RoboDK station: 15_holes_program_with_paths.rdk

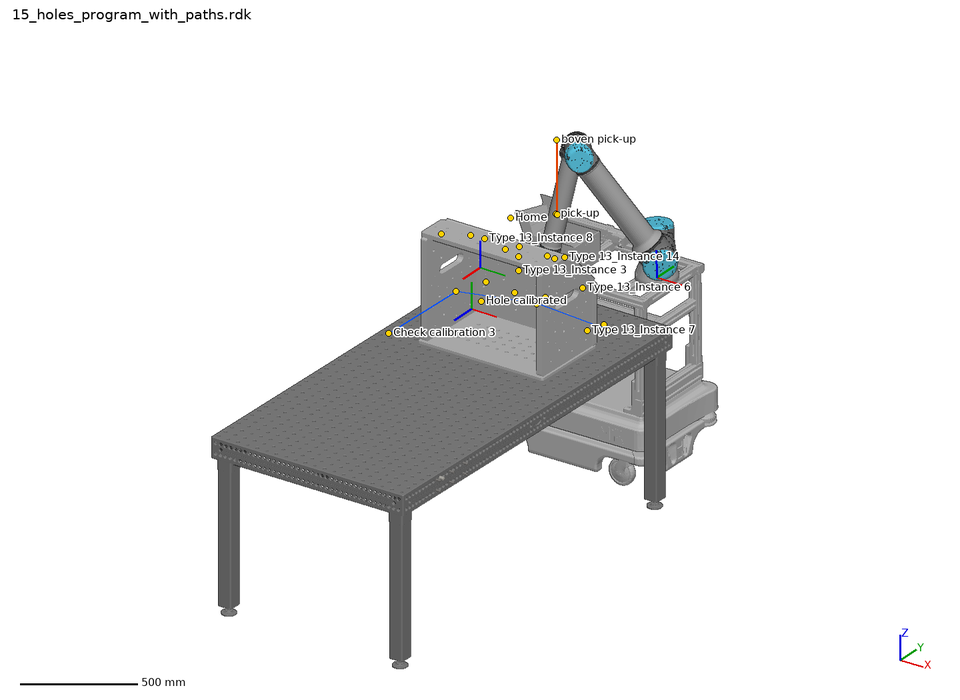
[picture v0: the station drawn from its stored meshes, robots at their saved joint values, targets as dots, program paths as lines]
Station 15_holes_program_with_paths (saved by RoboDK 5.7.0). Poses are relative to the parent item; angles as X-Y-Z fixed-axis rotations.
Station parameters (name, value as stored): 0.4, 1, 1, CollisionFreePlanner, UR10e, CollisionFreePlanner-Rob UR10e, Simplify-Mesh-Settings
  - object Lastafel at (0, 0, 0) mm, size 1021.8 x 2000 x 842 mm
  - object Lastafel_simplified at (0, 0, 0) mm, size 1000 x 2000 x 802.1 mm
  - frame UR10e Base at (-300.71, 2160.25, 91.6) mm, rotated rx 0.6 ry -0.16 rz 0.46 deg
    - robot UR10e: 6 axes, payload 10 kg, reach 1300 mm, repeatability 0.05 mm, weight 28.9 kg
        modified DH rows (alpha deg, a mm, theta deg, d mm): 0, 0, 0, 180.7; 90, 0, 180, 0; 0, 612.6, 0, 0; 0, 571.335, 0, 174.15; -90, 0, 0, 119.85; 90, 0, 180, 116.55
        joint limits [-70, -140, 0, -220, -180, -280] to [85, 0, 170, 200, 180, 115]; home [30.872, -95.296, 116.362, -22.187, 121.11, 179.827]; saved at [38.401, -56.267, 133.515, -77.437, 128.806, 0.409]
      - tool Screwdriver indraaitool, TCP at (215, -0.23, 99.66) mm, rotated rx 0 ry 90 rz 0 deg, size 345 x 117.4 x 144.9 mm, geometry from 0 Screwdriver assembly.STEP
      - tool Camera, TCP at (304, 50.7, 13.6) mm, rotated rx 0 ry 90 rz 0 deg
      - tool pointer, TCP at (196, -0.23, 99.66) mm, rotated rx 0 ry 90 rz 0 deg
      - tool Screwdriver simplified, TCP at (0, 0, 220) mm, size 159.8 x 129.1 x 379.7 mm, geometry from Screwdriver simplified.stl
      - tool indraaien, TCP at (205, 0.2, 100) mm, rotated rx 0 ry 90 rz 0 deg
    - object Assembly mir + frame aangepast naar ur10e versie 2 at (-733.08, 277.19, -552.66) mm, rotated rx 90 ry 0 rz 0.45 deg, size 901.1 x 1139.6 x 580.4 mm, geometry from Assembly mir + frame aangepast naar ur10e versie 2.STEP
    - object Mir + frame simplified at (-733.08, 277.19, -552.66) mm, rotated rx 90 ry 0 rz 0.45 deg, size 925.7 x 1139.7 x 582 mm
    - target boven pick-up (joint target) at (-657.55, 210.4, 385.42) mm, rotated rx 180 ry -0.01 rz 58.34 deg; joints [-50.868, -81.351, 94.607, -13.692, -19.23, -89.565] of UR10e
    - target pick-up (joint target) at (-663.21, 209.22, 32.36) mm, rotated rx 179.99 ry 0 rz 58.33 deg; joints [-50.468, -67.472, 110.452, -43.416, -18.832, -89.554] of UR10e
    - target unclamped (joint target) at (-658.69, 209.89, 32.4) mm, rotated rx -180 ry 0 rz 58.34 deg; joints [-50.794, -47.979, 113.128, 114.877, 19.182, -270.008] of UR10e
  - frame Hoek lastafel at (-1020, 1876.5, 50) mm, rotated rx 0 ry 0 rz -90 deg
    - frame CSV Frame at (350, 200, 0) mm, rotated rx 90 ry 0 rz 90 deg
      - object Test object at (0, 0.01, 0) mm, size 650 x 517 x 400 mm, geometry from Test object.STEP
      - object Test object simplified at (0, 0.01, 0) mm, size 650.1 x 517 x 436.5 mm
      - frame Type 13 at (0, 0, 0) mm
        - target Hole calibrated (Cartesian target) at (50, 50, 0) mm; joints [38.401, -56.267, 133.515, -77.437, 128.806, 0.409] of UR10e
        - target Type 13_Instance 2 (Cartesian target) at (224.21, 141.91, 0) mm, rotated rx 0 ry 0 rz 120 deg; joints [21.978, -61.024, 129.364, 49.468, 78.603, 19.537] of UR10e
        - target Type 13_Instance 3 (Cartesian target) at (246.01, 251.55, 0) mm, rotated rx 0 ry 0 rz 80 deg; joints [29.991, -83.076, 133.126, 30.949, 94.737, 30.232] of UR10e
        - target Type 13_Instance 5 (Cartesian target) at (382.2, 163.02, 0) mm, rotated rx 0 ry 0 rz 100 deg; joints [40.216, -73.928, 140.296, 30.8, 83.246, 40.29] of UR10e
        - target Type 13_Instance 6 (Cartesian target) at (577.65, 261.77, 0) mm, rotated rx 0 ry 0 rz 80 deg; joints [83.526, -84.373, 135.629, 37.157, 100.147, 84.01] of UR10e
        - target Type 13_Instance 7 (Cartesian target) at (602.84, 67, 0) mm, rotated rx 0 ry 0 rz 140 deg; joints [61.233, -52.023, 142.726, 28.243, 47.512, 50] of UR10e
        - target Type 13_Instance 8 (Cartesian target) at (128.87, 405.62, 85.34) mm, rotated rx 0 ry 45 rz -90 deg; joints [24.723, -96.328, 122.329, -93.279, 50.619, -33.648] of UR10e
        - target Type 13_Instance 10 (Cartesian target) at (325.68, 432.59, 112.3) mm, rotated rx 0 ry 45 rz -90 deg; joints [39.423, -108.608, 126.743, -75.897, 57.444, -49.793] of UR10e
        - target Type 13_Instance 12 (Cartesian target) at (502.06, 421.99, 101.71) mm, rotated rx 0 ry 45 rz -90 deg; joints [56.925, -115.887, 130.806, -65.302, 67.776, -65.755] of UR10e
        - target Type 13_Instance 13 (Cartesian target) at (570.16, 369.5, 49.22) mm, rotated rx 0 ry 45 rz -90 deg; joints [62.403, -121.656, 138.779, -65.954, 71.328, -70.219] of UR10e
        - target Type 13_Instance 14 (Cartesian target) at (588.54, 468.7, 148.42) mm, rotated rx 0 ry 45 rz -90 deg; joints [71.01, -111.335, 122.877, -58.584, 77.085, -76.834] of UR10e
        - target Type 13_Instance 15 (Cartesian target) at (192.89, 517, 279.7) mm, rotated rx 0 ry 90 rz -90 deg; joints [52.145, -62.069, 43.009, 18.396, 52.67, -89.759] of UR10e
        - target Type 13_Instance 16 (Cartesian target) at (83.93, 517, 343.03) mm, rotated rx 90 ry 80 rz 0 deg; joints [50.032, -46.238, 16.171, 29.419, 60.538, -89.707] of UR10e
        - target Type 13_Instance 17 (Cartesian target) at (391.06, 517, 308.3) mm, rotated rx 0 ry 90 rz -90 deg; joints [65.267, -66.64, 49.834, 16.228, 65.797, -89.935] of UR10e
        - target Type 13_Instance 18 (Cartesian target) at (577.65, 517, 262.67) mm, rotated rx 0 ry 90 rz -90 deg; joints [77.626, -73.739, 59.711, 13.488, 78.165, -90.075] of UR10e
        - target Type 13_Instance 19 (Cartesian target) at (479.58, 517, 336.9) mm, rotated rx 0 ry 90 rz -90 deg; joints [71.94, -64.785, 47.115, 17.114, 72.467, -90.001] of UR10e
    - target Camera -90 (Cartesian target) at (100, 100, 0) mm, rotated rx 180 ry 0 rz 90 deg; joints [15.382, -77.593, 120.955, -43.48, 105.947, -89.524] of UR10e
    - target Camera +90 (Cartesian target) at (100, 100, 0) mm, rotated rx -180 ry 0 rz -90 deg; joints [17.251, -55.937, 87.569, -31.877, -72.203, -90.48] of UR10e
    - target Camera Calibration (Cartesian target) at (100, 100, 0) mm, rotated rx -180 ry 0 rz 180 deg; joints [5.018, -68.171, 107.665, -44.191, 5.596, -85.486] of UR10e
    - target Camera 2 (Cartesian target) at (150, 750, 0) mm, rotated rx 180 ry 0 rz 180 deg; joints [50.749, -60.173, 157.418, 81.984, -51.264, -269.754] of UR10e
    - target Check calibration 0 (Cartesian target) at (200, 800, 10) mm, rotated rx 180 ry 0 rz 180 deg; joints [69.087, -96.044, 157.848, -62.324, 69.685, -90.102] of UR10e
    - target Check calibration 1 (Cartesian target) at (150, 400, 2) mm, rotated rx 180 ry 0 rz 180 deg; joints [4.739, -84.216, 147.782, -67.962, 5.34, -85.787] of UR10e
    - target Check calibration 2 (Cartesian target) at (250, 50, 2) mm, rotated rx 180 ry 0 rz 180 deg; joints [9.934, -58.947, 106.867, -51.902, 9.691, -86.238] of UR10e
    - target Check calibration 3 (Cartesian target) at (750, 50, 2) mm, rotated rx 180 ry 0 rz 180 deg; joints [40.424, -35.05, 60.293, -26.389, 40.152, -89.277] of UR10e
    - target Home (Cartesian target) at (200, 300, 400) mm, rotated rx 180 ry 0 rz 180 deg; joints [9.713, -85.986, 130.341, 132.467, -10.3, 92.957] of UR10e
  - program Check XY-calibration (7 instructions, listed below)
  - program bovenpickupToType13Instance2 (10 instructions, listed below)
  - program bovenpickupToType13Instance3 (10 instructions, listed below)
  - program bovenpickupToType13Instance5 (11 instructions, listed below)
  - program bovenpickupToType13Instance6 (10 instructions, listed below)
  - program bovenpickupToType13Instance7 (10 instructions, listed below)
  - program bovenpickupToType13Instance8 (12 instructions, listed below)
  - program bovenpickupToType13Instance10 (12 instructions, listed below)
  - program bovenpickupToType13Instance12 (13 instructions, listed below)
  - program bovenpickupToType13Instance13 (13 instructions, listed below)
  - program bovenpickupToType13Instance14 (16 instructions, listed below)
  - program bovenpickupToType13Instance15 (9 instructions, listed below)
  - program bovenpickupToType13Instance16 (13 instructions, listed below)
  - program bovenpickupToType13Instance17 (10 instructions, listed below)
  - program bovenpickupToType13Instance18 (11 instructions, listed below)
  - program bovenpickupToType13Instance19 (11 instructions, listed below)
  - program Type13Instance2Tobovenpickup (11 instructions, listed below)
  - program Type13Instance3Tobovenpickup (10 instructions, listed below)
  - program Type13Instance5Tobovenpickup (12 instructions, listed below)
  - program Type13Instance6Tobovenpickup (10 instructions, listed below)
  - program Type13Instance7Tobovenpickup (12 instructions, listed below)
  - program Type13Instance8Tobovenpickup (14 instructions, listed below)
  - program Type13Instance10Tobovenpickup (11 instructions, listed below)
  - program Type13Instance12Tobovenpickup (12 instructions, listed below)
  - program Type13Instance13Tobovenpickup (11 instructions, listed below)
  - program Type13Instance14Tobovenpickup (11 instructions, listed below)
  - program Type13Instance15Tobovenpickup (9 instructions, listed below)
  - program Type13Instance16Tobovenpickup (10 instructions, listed below)
  - program Type13Instance17Tobovenpickup (10 instructions, listed below)
  - program Type13Instance18Tobovenpickup (10 instructions, listed below)
  - program Type13Instance19Tobovenpickup (10 instructions, listed below)
  - program helicoil pickup (9 instructions, listed below)
  - Python program retract shank (listed below)
  - Python program get_helicoil (listed below)
  - Python program Insert helicoil (listed below)
  - Python program pickup helicoil (listed below)
  - Python program Test get screwdriver data (listed below)
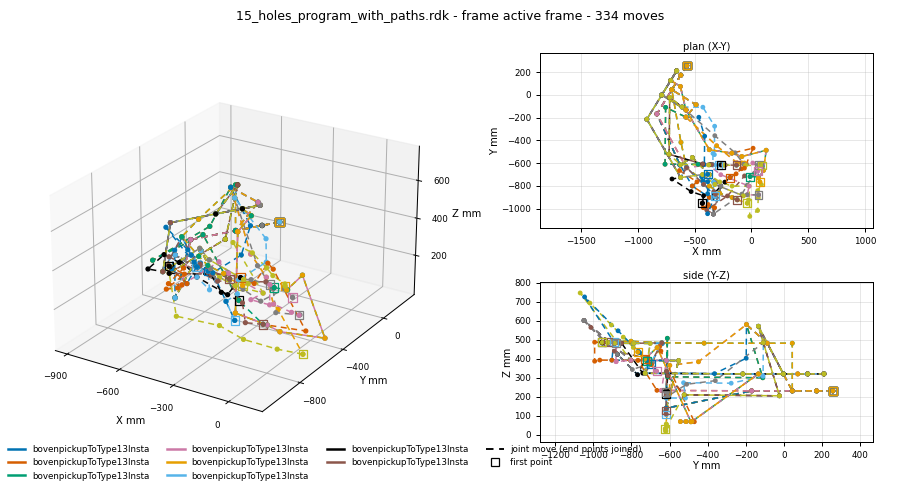
[picture p0: tool path of 15_holes_program_with_paths.rdk in frame active frame, 334 of 342 moves have a stored position in this frame; points joined in program order, loops and branches not executed]
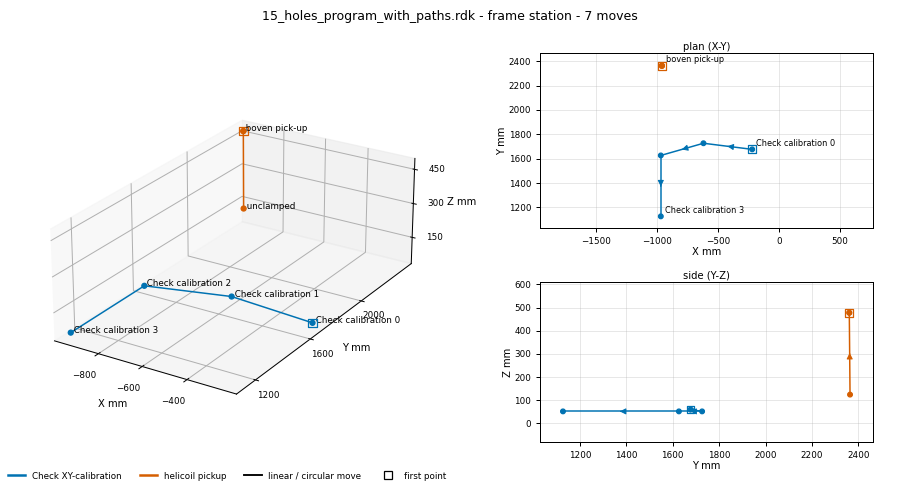
[picture p1: tool path of 15_holes_program_with_paths.rdk in frame station, 7 of 342 moves have a stored position in this frame; points joined in program order, loops and branches not executed]

--- program Check XY-calibration (robot UR10e) ---
  Set Ref.: Hoek lastafel
  Set Tool: pointer
  Set speed (200.0 mm/s)
  MoveL (Check calibration 0)
  MoveL (Check calibration 1)
  MoveL (Check calibration 2)
  MoveL (Check calibration 3)

--- program bovenpickupToType13Instance2 (robot UR10e) ---
  MoveJ (Pt 1 (S642)) to (-569.02, 256.95, 231.44) mm, rotated rx 180 ry -0.01 rz 58.34 deg; joints [-50.868, -81.351, 94.607, -13.692, -19.23, -89.565]
  MoveJ (Pt 2 (S577)) to (-621.5, 171.83, 231.42) mm, rotated rx 180 ry -0.01 rz 58.34 deg; joints [-42.328, -81.409, 94.677, -14.057, -10.69, -89.211]
  MoveJ (Pt 3 (S442)) to (-700.22, 44.15, 231.39) mm, rotated rx 180 ry -0.01 rz 58.34 deg; joints [-29.369, -77.97, 90.586, -9.022, 2.264, -93.593]
  MoveJ (Pt 4 (S421)) to (-487.45, -87.1, 481.39) mm, rotated rx 180 ry -0.01 rz 58.34 deg; joints [-28.022, -101.389, 88.85, 14.844, 3.631, -92.304]
  MoveJ (Pt 5 (S124)) to (-576.74, -196.35, 579.46) mm, rotated rx 89.55 ry -40 rz 0.16 deg; joints [-35.971, -95.179, 103.829, 37.546, 63.204, -24.789]
  MoveJ (Pt 6 (S114)) to (-462.71, -197.66, 402.38) mm, rotated rx 88.03 ry -79.99 rz 1.82 deg; joints [-40.872, -92.425, 119.324, 55.78, 83.328, -40.3]
  MoveJ (Pt 7 (S42)) to (-411.56, -364.05, 321.78) mm, rotated rx -88.79 ry -60.15 rz 178.37 deg; joints [-15.974, -82.156, 125.219, 76.084, 97.176, -13.671]
  MoveJ (Pt 8 (S10)) to (-414.11, -614.03, 324.41) mm, rotated rx -88.79 ry -60.15 rz 178.37 deg; joints [16.405, -73.929, 114.079, 78.537, 81.219, 14.568]
  MoveJ (Pt 9 (S23)) to (-339.48, -616.15, 194.31) mm, rotated rx -88.79 ry -60.15 rz 178.37 deg; joints [19.42, -67.896, 124.439, 61.697, 79.797, 17.249]
  MoveJ (Pt 10 (S33)) to (-289.72, -617.57, 107.58) mm, rotated rx -88.79 ry -60.15 rz 178.37 deg; joints [21.978, -61.024, 129.364, 49.468, 78.603, 19.537]

--- program bovenpickupToType13Instance3 (robot UR10e) ---
  MoveJ (Pt 1 (S258)) to (-569.02, 256.95, 231.44) mm, rotated rx 180 ry -0.01 rz 58.34 deg; joints [-50.868, -81.351, 94.607, -13.692, -19.23, -89.565]
  MoveJ (Pt 2 (S259)) to (-621.5, 171.83, 231.42) mm, rotated rx 180 ry -0.01 rz 58.34 deg; joints [-42.328, -81.409, 94.677, -14.057, -10.69, -89.211]
  MoveJ (Pt 3 (S230)) to (-700.22, 44.15, 231.39) mm, rotated rx 180 ry -0.01 rz 58.34 deg; joints [-29.369, -77.97, 90.586, -9.022, 2.264, -93.593]
  MoveJ (Pt 4 (S386)) to (-487.45, -87.1, 481.39) mm, rotated rx 180 ry -0.01 rz 58.34 deg; joints [-28.022, -101.389, 88.85, 14.844, 3.631, -92.304]
  MoveJ (Pt 5 (S758)) to (-576.74, -196.35, 579.46) mm, rotated rx 89.55 ry -40 rz 0.16 deg; joints [-35.971, -95.179, 103.829, 37.546, 63.204, -24.789]
  MoveJ (Pt 6 (S704)) to (-754.66, -110.75, 300.04) mm, rotated rx 86.59 ry -79.83 rz 2.77 deg; joints [-30.172, -60.169, 89.434, 52.244, 84.533, -29.177]
  MoveJ (Pt 7 (S702)) to (-759.76, -610.7, 305.28) mm, rotated rx 86.59 ry -79.83 rz 2.77 deg; joints [10.723, -56.863, 83.085, 53.769, 91.432, 11.188]
  MoveJ (Pt 8 (S856)) to (-469.6, -611.54, 507.29) mm, rotated rx 86.59 ry -79.83 rz 2.77 deg; joints [17.574, -86.724, 101.894, 65.055, 92.657, 17.965]
  MoveJ (Pt 9 (S864)) to (-348.42, -614.6, 333.21) mm, rotated rx 86.59 ry -79.83 rz 2.77 deg; joints [23.724, -87.864, 122.531, 45.887, 93.715, 24.039]
  MoveJ (Pt 10 (S846)) to (-267.62, -616.65, 217.16) mm, rotated rx 86.59 ry -79.83 rz 2.77 deg; joints [29.991, -83.076, 133.126, 30.949, 94.737, 30.232]

--- program bovenpickupToType13Instance5 (robot UR10e) ---
  MoveJ (Pt 1 (S221)) to (-569.02, 256.95, 231.44) mm, rotated rx 180 ry -0.01 rz 58.34 deg; joints [-50.868, -81.351, 94.607, -13.692, -19.23, -89.565]
  MoveJ (Pt 2 (S222)) to (-621.5, 171.83, 231.42) mm, rotated rx 180 ry -0.01 rz 58.34 deg; joints [-42.328, -81.409, 94.677, -14.057, -10.69, -89.211]
  MoveJ (Pt 3 (S200)) to (-700.22, 44.15, 231.39) mm, rotated rx 180 ry -0.01 rz 58.34 deg; joints [-29.369, -77.97, 90.586, -9.022, 2.264, -93.593]
  MoveJ (Pt 4 (S356)) to (-487.45, -87.1, 481.39) mm, rotated rx 180 ry -0.01 rz 58.34 deg; joints [-28.022, -101.389, 88.85, 14.844, 3.631, -92.304]
  MoveJ (Pt 5 (S742)) to (-576.74, -196.35, 579.46) mm, rotated rx 89.55 ry -40 rz 0.16 deg; joints [-35.971, -95.179, 103.829, 37.546, 63.204, -24.789]
  MoveJ (Pt 6 (S692)) to (-754.66, -110.75, 300.04) mm, rotated rx 86.59 ry -79.83 rz 2.77 deg; joints [-30.172, -60.169, 89.434, 52.244, 84.533, -29.177]
  MoveJ (Pt 7 (S687)) to (-759.76, -610.7, 305.28) mm, rotated rx 86.59 ry -79.83 rz 2.77 deg; joints [10.723, -56.863, 83.085, 53.769, 91.432, 11.188]
  MoveJ (Pt 8 (S846)) to (-469.6, -611.54, 507.29) mm, rotated rx 86.59 ry -79.83 rz 2.77 deg; joints [17.574, -86.724, 101.894, 65.055, 92.657, 17.965]
  MoveJ (Pt 9 (S855)) to (-348.42, -614.6, 333.21) mm, rotated rx 86.59 ry -79.83 rz 2.77 deg; joints [23.724, -87.864, 122.531, 45.887, 93.715, 24.039]
  MoveJ (Pt 10 (S832)) to (-267.62, -616.65, 217.16) mm, rotated rx 86.59 ry -79.83 rz 2.77 deg; joints [29.991, -83.076, 133.126, 30.949, 94.737, 30.232]
  MoveJ (Pt 11 (S795)) to (-131.68, -618.97, 128.27) mm, rotated rx -86.49 ry -80.13 rz 175.95 deg; joints [40.216, -73.928, 140.296, 30.8, 83.246, 40.29]

--- program bovenpickupToType13Instance6 (robot UR10e) ---
  MoveJ (Pt 1 (S198)) to (-569.02, 256.95, 231.44) mm, rotated rx 180 ry -0.01 rz 58.34 deg; joints [-50.868, -81.351, 94.607, -13.692, -19.23, -89.565]
  MoveJ (Pt 2 (S200)) to (-621.5, 171.83, 231.42) mm, rotated rx 180 ry -0.01 rz 58.34 deg; joints [-42.328, -81.409, 94.677, -14.057, -10.69, -89.211]
  MoveJ (Pt 3 (S176)) to (-700.22, 44.15, 231.39) mm, rotated rx 180 ry -0.01 rz 58.34 deg; joints [-29.369, -77.97, 90.586, -9.022, 2.264, -93.593]
  MoveJ (Pt 4 (S337)) to (-487.45, -87.1, 481.39) mm, rotated rx 180 ry -0.01 rz 58.34 deg; joints [-28.022, -101.389, 88.85, 14.844, 3.631, -92.304]
  MoveJ (Pt 5 (S753)) to (-576.74, -196.35, 579.46) mm, rotated rx 89.55 ry -40 rz 0.16 deg; joints [-35.971, -95.179, 103.829, 37.546, 63.204, -24.789]
  MoveJ (Pt 6 (S927)) to (-306.31, -448.13, 384.07) mm, rotated rx 89.47 ry -50 rz 0.28 deg; joints [-10.312, -118.158, 138.236, 30.476, 83.322, -7.663]
  MoveJ (Pt 7 (S951)) to (-127.46, -598.64, 365.16) mm, rotated rx 89.47 ry -50 rz 0.28 deg; joints [52.736, -103.918, 134.566, 32.325, 120.747, 45.438]
  MoveJ (Pt 8 (S904)) to (-87.05, -599.5, 236.84) mm, rotated rx 88.03 ry -79.99 rz 1.82 deg; joints [51.039, -92.195, 140.398, 35.287, 97.676, 50.753]
  MoveJ (Pt 9 (S953)) to (11.43, -599.82, 219.48) mm, rotated rx 88.03 ry -79.99 rz 1.82 deg; joints [71.326, -88.12, 140.046, 34.604, 99.482, 71.185]
  MoveJ (Pt 10 (S985)) to (64.03, -619.93, 226.49) mm, rotated rx 86.59 ry -79.83 rz 2.77 deg; joints [83.526, -84.373, 135.629, 37.157, 100.147, 84.01]

--- program bovenpickupToType13Instance7 (robot UR10e) ---
  MoveJ (Pt 1 (S624)) to (-569.02, 256.95, 231.44) mm, rotated rx 180 ry -0.01 rz 58.34 deg; joints [-50.868, -81.351, 94.607, -13.692, -19.23, -89.565]
  MoveJ (Pt 2 (S566)) to (-621.5, 171.83, 231.42) mm, rotated rx 180 ry -0.01 rz 58.34 deg; joints [-42.328, -81.409, 94.677, -14.057, -10.69, -89.211]
  MoveJ (Pt 3 (S508)) to (-700.22, 44.15, 231.39) mm, rotated rx 180 ry -0.01 rz 58.34 deg; joints [-29.369, -77.97, 90.586, -9.022, 2.264, -93.593]
  MoveJ (Pt 4 (S484)) to (-487.45, -87.1, 481.39) mm, rotated rx 180 ry -0.01 rz 58.34 deg; joints [-28.022, -101.389, 88.85, 14.844, 3.631, -92.304]
  MoveJ (Pt 5 (S95)) to (-576.74, -196.35, 579.46) mm, rotated rx 89.55 ry -40 rz 0.16 deg; joints [-35.971, -95.179, 103.829, 37.546, 63.204, -24.789]
  MoveJ (Pt 6 (S69)) to (-306.31, -448.13, 384.07) mm, rotated rx 89.47 ry -50 rz 0.28 deg; joints [-10.312, -118.158, 138.236, 30.476, 83.322, -7.663]
  MoveJ (Pt 7 (S117)) to (-127.46, -598.64, 365.16) mm, rotated rx 89.47 ry -50 rz 0.28 deg; joints [52.736, -103.918, 134.566, 32.325, 120.747, 45.438]
  MoveJ (Pt 8 (S81)) to (-87.05, -599.5, 236.84) mm, rotated rx 88.03 ry -79.99 rz 1.82 deg; joints [51.039, -92.195, 140.398, 35.287, 97.676, 50.753]
  MoveJ (Pt 9 (S67)) to (-61.73, -599.68, 215.66) mm, rotated rx -0.06 ry -89.66 rz 89.93 deg; joints [51.732, -89.449, 141.404, 37.841, 89.906, 51.849]
  MoveJ (Pt 10 (S129)) to (88.68, -622.23, 31.67) mm, rotated rx -89.21 ry -40.15 rz 178.91 deg; joints [61.233, -52.023, 142.726, 28.243, 47.512, 50]

--- program bovenpickupToType13Instance8 (robot UR10e) ---
  MoveJ (Pt 1 (S440)) to (-569.02, 256.95, 231.44) mm, rotated rx 180 ry -0.01 rz 58.34 deg; joints [-50.868, -81.351, 94.607, -13.692, -19.23, -89.565]
  MoveJ (Pt 2 (S437)) to (-621.5, 171.83, 231.42) mm, rotated rx 180 ry -0.01 rz 58.34 deg; joints [-42.328, -81.409, 94.677, -14.057, -10.69, -89.211]
  MoveJ (Pt 3 (S490)) to (-700.22, 44.15, 231.39) mm, rotated rx 180 ry -0.01 rz 58.34 deg; joints [-29.369, -77.97, 90.586, -9.022, 2.264, -93.593]
  MoveJ (Pt 4 (S533)) to (-831.43, -168.65, 231.34) mm, rotated rx 180 ry -0.01 rz 58.34 deg; joints [-10.139, -68.333, 77.878, -9.215, 21.482, -90.324]
  MoveJ (Pt 5 (S587)) to (-628.82, -616.83, 140.7) mm, rotated rx 180 ry 0.34 rz 89.87 deg; joints [23.562, -63.896, 80.895, -17.582, 23.654, -89.485]
  MoveJ (Pt 6 (S610)) to (-519.72, -552.25, 390.32) mm, rotated rx 180 ry 0.34 rz 89.87 deg; joints [22.274, -79.112, 75.978, 2.531, 22.373, -89.461]
  MoveJ (Pt 7 (S617)) to (-370.06, -702.58, 391.22) mm, rotated rx 180 ry 0.34 rz 89.87 deg; joints [39.494, -78.996, 75.747, 2.876, 39.592, -89.745]
  MoveJ (Pt 8 (S629)) to (-270.28, -802.8, 391.81) mm, rotated rx 180 ry 0.34 rz 89.87 deg; joints [50.999, -75.487, 71.344, 3.823, 51.092, -89.834]
  MoveJ (Pt 9 (S393)) to (-334.84, -1048.74, 600.68) mm, rotated rx 180 ry 45.34 rz 89.87 deg; joints [50.594, -75.677, 73.548, -50.385, 63.524, -59.847]
  MoveJ (Pt 10 (S181)) to (-334.45, -873.03, 422.85) mm, rotated rx 180 ry 45.34 rz 89.87 deg; joints [41.069, -88.108, 106.775, -75.506, 58, -50.992]
  MoveJ (Pt 11 (S109)) to (-334.21, -767.6, 316.15) mm, rotated rx 180 ry 45.34 rz 89.87 deg; joints [33.25, -91.757, 123.172, -92.767, 53.974, -42.917]
  MoveJ (Pt 12 (S94)) to (-385.19, -699.16, 372.43) mm, rotated rx -179.78 ry 45.6 rz 89.57 deg; joints [24.723, -96.328, 122.329, -93.279, 50.619, -33.648]

--- program bovenpickupToType13Instance10 (robot UR10e) ---
  MoveJ (Pt 1 (S435)) to (-569.02, 256.95, 231.44) mm, rotated rx 180 ry -0.01 rz 58.34 deg; joints [-50.868, -81.351, 94.607, -13.692, -19.23, -89.565]
  MoveJ (Pt 2 (S375)) to (-621.5, 171.83, 231.42) mm, rotated rx 180 ry -0.01 rz 58.34 deg; joints [-42.328, -81.409, 94.677, -14.057, -10.69, -89.211]
  MoveJ (Pt 3 (S354)) to (-700.22, 44.15, 231.39) mm, rotated rx 180 ry -0.01 rz 58.34 deg; joints [-29.369, -77.97, 90.586, -9.022, 2.264, -93.593]
  MoveJ (Pt 4 (S390)) to (-831.43, -168.65, 231.34) mm, rotated rx 180 ry -0.01 rz 58.34 deg; joints [-10.139, -68.333, 77.878, -9.215, 21.482, -90.324]
  MoveJ (Pt 5 (S468)) to (-628.82, -616.83, 140.7) mm, rotated rx 180 ry 0.34 rz 89.87 deg; joints [23.562, -63.896, 80.895, -17.582, 23.654, -89.485]
  MoveJ (Pt 6 (S551)) to (-519.72, -552.25, 390.32) mm, rotated rx 180 ry 0.34 rz 89.87 deg; joints [22.274, -79.112, 75.978, 2.531, 22.373, -89.461]
  MoveJ (Pt 7 (S554)) to (-370.06, -702.58, 391.22) mm, rotated rx 180 ry 0.34 rz 89.87 deg; joints [39.494, -78.996, 75.747, 2.876, 39.592, -89.745]
  MoveJ (Pt 8 (S563)) to (-270.28, -802.8, 391.81) mm, rotated rx 180 ry 0.34 rz 89.87 deg; joints [50.999, -75.487, 71.344, 3.823, 51.092, -89.834]
  MoveJ (Pt 9 (S276)) to (-334.84, -1048.74, 600.68) mm, rotated rx 180 ry 45.34 rz 89.87 deg; joints [50.594, -75.677, 73.548, -50.385, 63.524, -59.847]
  MoveJ (Pt 10 (S138)) to (-334.45, -873.03, 422.85) mm, rotated rx 180 ry 45.34 rz 89.87 deg; joints [41.069, -88.108, 106.775, -75.506, 58, -50.992]
  MoveJ (Pt 11 (S166)) to (-234.21, -767.82, 316.15) mm, rotated rx 180 ry 45.34 rz 89.87 deg; joints [39.518, -97.83, 127.836, -87.655, 57.153, -49.479]
  MoveJ (Pt 12 (S207)) to (-188.6, -727.86, 399.15) mm, rotated rx -179.78 ry 45.6 rz 89.57 deg; joints [39.423, -108.608, 126.743, -75.897, 57.444, -49.793]

--- program bovenpickupToType13Instance12 (robot UR10e) ---
  MoveJ (Pt 1 (S490)) to (-569.02, 256.95, 231.44) mm, rotated rx 180 ry -0.01 rz 58.34 deg; joints [-50.868, -81.351, 94.607, -13.692, -19.23, -89.565]
  MoveJ (Pt 2 (S451)) to (-621.5, 171.83, 231.42) mm, rotated rx 180 ry -0.01 rz 58.34 deg; joints [-42.328, -81.409, 94.677, -14.057, -10.69, -89.211]
  MoveJ (Pt 3 (S503)) to (-700.22, 44.15, 231.39) mm, rotated rx 180 ry -0.01 rz 58.34 deg; joints [-29.369, -77.97, 90.586, -9.022, 2.264, -93.593]
  MoveJ (Pt 4 (S564)) to (-831.43, -168.65, 231.34) mm, rotated rx 180 ry -0.01 rz 58.34 deg; joints [-10.139, -68.333, 77.878, -9.215, 21.482, -90.324]
  MoveJ (Pt 5 (S627)) to (-628.82, -616.83, 140.7) mm, rotated rx 180 ry 0.34 rz 89.87 deg; joints [23.562, -63.896, 80.895, -17.582, 23.654, -89.485]
  MoveJ (Pt 6 (S652)) to (-519.72, -552.25, 390.32) mm, rotated rx 180 ry 0.34 rz 89.87 deg; joints [22.274, -79.112, 75.978, 2.531, 22.373, -89.461]
  MoveJ (Pt 7 (S659)) to (-370.06, -702.58, 391.22) mm, rotated rx 180 ry 0.34 rz 89.87 deg; joints [39.494, -78.996, 75.747, 2.876, 39.592, -89.745]
  MoveJ (Pt 8 (S674)) to (-270.28, -802.8, 391.81) mm, rotated rx 180 ry 0.34 rz 89.87 deg; joints [50.999, -75.487, 71.344, 3.823, 51.092, -89.834]
  MoveJ (Pt 9 (S406)) to (-334.84, -1048.74, 600.68) mm, rotated rx 180 ry 45.34 rz 89.87 deg; joints [50.594, -75.677, 73.548, -50.385, 63.524, -59.847]
  MoveJ (Pt 10 (S321)) to (-393.48, -1012.72, 564.35) mm, rotated rx 180 ry 45.34 rz 89.87 deg; joints [45.833, -76.136, 78.115, -56.513, 60.695, -55.521]
  MoveJ (Pt 11 (S226)) to (-211.3, -889.58, 439.32) mm, rotated rx 180 ry 45.34 rz 89.87 deg; joints [50.01, -92.787, 108.942, -68.876, 63.158, -59.384]
  MoveJ (Pt 12 (S275)) to (-60.91, -713.35, 402.9) mm, rotated rx 180 ry 45.34 rz 89.87 deg; joints [50.234, -115.862, 129.495, -66.244, 63.307, -59.629]
  MoveJ (Pt 13 (S348)) to (-12.15, -719.18, 387.98) mm, rotated rx -179.78 ry 45.6 rz 89.57 deg; joints [56.925, -115.887, 130.806, -65.302, 67.776, -65.755]

--- program bovenpickupToType13Instance13 (robot UR10e) ---
  MoveJ (Pt 1 (S502)) to (-569.02, 256.95, 231.44) mm, rotated rx 180 ry -0.01 rz 58.34 deg; joints [-50.868, -81.351, 94.607, -13.692, -19.23, -89.565]
  MoveJ (Pt 2 (S497)) to (-621.5, 171.83, 231.42) mm, rotated rx 180 ry -0.01 rz 58.34 deg; joints [-42.328, -81.409, 94.677, -14.057, -10.69, -89.211]
  MoveJ (Pt 3 (S556)) to (-700.22, 44.15, 231.39) mm, rotated rx 180 ry -0.01 rz 58.34 deg; joints [-29.369, -77.97, 90.586, -9.022, 2.264, -93.593]
  MoveJ (Pt 4 (S613)) to (-831.43, -168.65, 231.34) mm, rotated rx 180 ry -0.01 rz 58.34 deg; joints [-10.139, -68.333, 77.878, -9.215, 21.482, -90.324]
  MoveJ (Pt 5 (S672)) to (-628.82, -616.83, 140.7) mm, rotated rx 180 ry 0.34 rz 89.87 deg; joints [23.562, -63.896, 80.895, -17.582, 23.654, -89.485]
  MoveJ (Pt 6 (S701)) to (-519.72, -552.25, 390.32) mm, rotated rx 180 ry 0.34 rz 89.87 deg; joints [22.274, -79.112, 75.978, 2.531, 22.373, -89.461]
  MoveJ (Pt 7 (S705)) to (-370.06, -702.58, 391.22) mm, rotated rx 180 ry 0.34 rz 89.87 deg; joints [39.494, -78.996, 75.747, 2.876, 39.592, -89.745]
  MoveJ (Pt 8 (S722)) to (-270.28, -802.8, 391.81) mm, rotated rx 180 ry 0.34 rz 89.87 deg; joints [50.999, -75.487, 71.344, 3.823, 51.092, -89.834]
  MoveJ (Pt 9 (S435)) to (-334.84, -1048.74, 600.68) mm, rotated rx 180 ry 45.34 rz 89.87 deg; joints [50.594, -75.677, 73.548, -50.385, 63.524, -59.847]
  MoveJ (Pt 10 (S331)) to (-84.45, -873.59, 422.85) mm, rotated rx 180 ry 45.34 rz 89.87 deg; joints [59.234, -97.73, 114.561, -66.365, 68.949, -67.251]
  MoveJ (Pt 11 (S272)) to (-37.47, -795.07, 343.28) mm, rotated rx 180 ry 45.34 rz 89.87 deg; joints [59.221, -104.089, 128.071, -73.512, 68.939, -67.26]
  MoveJ (Pt 12 (S398)) to (25.63, -689.69, 378.76) mm, rotated rx 180 ry 45.34 rz 89.87 deg; joints [59.247, -119.903, 133.427, -63.039, 68.975, -67.299]
  MoveJ (Pt 13 (S436)) to (56.33, -667.94, 334.76) mm, rotated rx -179.78 ry 45.6 rz 89.57 deg; joints [62.403, -121.656, 138.779, -65.954, 71.328, -70.219]

--- program bovenpickupToType13Instance14 (robot UR10e) ---
  MoveJ (Pt 1 (S636)) to (-569.02, 256.95, 231.44) mm, rotated rx 180 ry -0.01 rz 58.34 deg; joints [-50.868, -81.351, 94.607, -13.692, -19.23, -89.565]
  MoveJ (Pt 2 (S579)) to (-621.5, 171.83, 231.42) mm, rotated rx 180 ry -0.01 rz 58.34 deg; joints [-42.328, -81.409, 94.677, -14.057, -10.69, -89.211]
  MoveJ (Pt 3 (S532)) to (-700.22, 44.15, 231.39) mm, rotated rx 180 ry -0.01 rz 58.34 deg; joints [-29.369, -77.97, 90.586, -9.022, 2.264, -93.593]
  MoveJ (Pt 4 (S413)) to (-831.43, -168.65, 231.34) mm, rotated rx 180 ry -0.01 rz 58.34 deg; joints [-10.139, -68.333, 77.878, -9.215, 21.482, -90.324]
  MoveJ (Pt 5 (S470)) to (-628.82, -616.83, 140.7) mm, rotated rx 180 ry 0.34 rz 89.87 deg; joints [23.562, -63.896, 80.895, -17.582, 23.654, -89.485]
  MoveJ (Pt 6 (S573)) to (-519.72, -552.25, 390.32) mm, rotated rx 180 ry 0.34 rz 89.87 deg; joints [22.274, -79.112, 75.978, 2.531, 22.373, -89.461]
  MoveJ (Pt 7 (S576)) to (-370.06, -702.58, 391.22) mm, rotated rx 180 ry 0.34 rz 89.87 deg; joints [39.494, -78.996, 75.747, 2.876, 39.592, -89.745]
  MoveJ (Pt 8 (S593)) to (-279.16, -766.12, 391.6) mm, rotated rx 180 ry 0.34 rz 89.87 deg; joints [48.532, -78.392, 74.978, 3.089, 48.628, -89.822]
  MoveJ (Pt 9 (S651)) to (-170.28, -803.03, 391.82) mm, rotated rx 180 ry 0.34 rz 89.87 deg; joints [57.613, -79.202, 75.935, 2.972, 57.71, -89.885]
  MoveJ (Pt 10 (S740)) to (-20.28, -803.36, 391.82) mm, rotated rx 180 ry 0.34 rz 89.87 deg; joints [69.118, -82.29, 79.557, 2.458, 69.22, -89.954]
  MoveJ (Pt 11 (S665)) to (-14.78, -1068.99, 745.22) mm, rotated rx -179.78 ry 45.6 rz 89.57 deg; joints [72.225, -79.746, 63.029, -30.149, 77.907, -77.653]
  MoveJ (Pt 12 (S660)) to (53.7, -1017.76, 692.01) mm, rotated rx -179.78 ry 45.6 rz 89.57 deg; joints [76.38, -86.273, 75.842, -35.866, 80.759, -80.743]
  MoveJ (Pt 13 (S562)) to (60.07, -905.32, 577.11) mm, rotated rx -179.78 ry 45.6 rz 89.57 deg; joints [74.313, -98.133, 98.844, -47.262, 79.338, -79.258]
  MoveJ (Pt 14 (S517)) to (55.02, -842.85, 513.38) mm, rotated rx -179.78 ry 45.6 rz 89.57 deg; joints [71.837, -104.176, 110.096, -52.832, 77.645, -77.435]
  MoveJ (Pt 15 (S506)) to (87.31, -790.16, 459.16) mm, rotated rx -179.78 ry 45.6 rz 89.57 deg; joints [73.635, -108.918, 118.831, -56.552, 78.877, -78.786]
  MoveJ (Pt 16 (S476)) to (73.98, -766.28, 434.94) mm, rotated rx -179.78 ry 45.6 rz 89.57 deg; joints [71.01, -111.335, 122.877, -58.584, 77.085, -76.834]

--- program bovenpickupToType13Instance15 (robot UR10e) ---
  MoveJ (Pt 1 (S586)) to (-569.02, 256.95, 231.44) mm, rotated rx 180 ry -0.01 rz 58.34 deg; joints [-50.868, -81.351, 94.607, -13.692, -19.23, -89.565]
  MoveJ (Pt 2 (S526)) to (-621.5, 171.83, 231.42) mm, rotated rx 180 ry -0.01 rz 58.34 deg; joints [-42.328, -81.409, 94.677, -14.057, -10.69, -89.211]
  MoveJ (Pt 3 (S493)) to (-700.22, 44.15, 231.39) mm, rotated rx 180 ry -0.01 rz 58.34 deg; joints [-29.369, -77.97, 90.586, -9.022, 2.264, -93.593]
  MoveJ (Pt 4 (S423)) to (-831.43, -168.65, 231.34) mm, rotated rx 180 ry -0.01 rz 58.34 deg; joints [-10.139, -68.333, 77.878, -9.215, 21.482, -90.324]
  MoveJ (Pt 5 (S303)) to (-628.82, -616.83, 140.7) mm, rotated rx 180 ry 0.34 rz 89.87 deg; joints [23.562, -63.896, 80.895, -17.582, 23.654, -89.485]
  MoveJ (Pt 6 (S431)) to (-628.82, -615.34, 390.69) mm, rotated rx 180 ry 0.34 rz 89.87 deg; joints [23.488, -66.086, 58.723, 6.733, 23.569, -89.434]
  MoveJ (Pt 7 (S390)) to (-520.28, -802.24, 391.81) mm, rotated rx 180 ry 0.34 rz 89.87 deg; joints [38.28, -60.592, 50.44, 9.726, 38.353, -89.675]
  MoveJ (Pt 8 (S324)) to (-370.5, -902.58, 392.41) mm, rotated rx 180 ry 0.34 rz 89.87 deg; joints [50.012, -60.823, 50.732, 9.743, 50.085, -89.789]
  MoveJ (Pt 9 (S347)) to (-322.86, -892.99, 485.67) mm, rotated rx -179.85 ry 0.6 rz 89.42 deg; joints [52.145, -62.069, 43.009, 18.396, 52.67, -89.759]

--- program bovenpickupToType13Instance16 (robot UR10e) ---
  MoveJ (Pt 1 (S521)) to (-569.02, 256.95, 231.44) mm, rotated rx 180 ry -0.01 rz 58.34 deg; joints [-50.868, -81.351, 94.607, -13.692, -19.23, -89.565]
  MoveJ (Pt 2 (S472)) to (-621.5, 171.83, 231.42) mm, rotated rx 180 ry -0.01 rz 58.34 deg; joints [-42.328, -81.409, 94.677, -14.057, -10.69, -89.211]
  MoveJ (Pt 3 (S342)) to (-700.22, 44.15, 231.39) mm, rotated rx 180 ry -0.01 rz 58.34 deg; joints [-29.369, -77.97, 90.586, -9.022, 2.264, -93.593]
  MoveJ (Pt 4 (S284)) to (-831.43, -168.65, 231.34) mm, rotated rx 180 ry -0.01 rz 58.34 deg; joints [-10.139, -68.333, 77.878, -9.215, 21.482, -90.324]
  MoveJ (Pt 5 (S181)) to (-570.99, -643.08, 233.72) mm, rotated rx -179.85 ry 0.6 rz 89.42 deg; joints [26.976, -69.099, 78.835, -10.802, 27.531, -89.229]
  MoveJ (Pt 6 (S175)) to (-632.97, -666.16, 234.14) mm, rotated rx -179.95 ry 0.62 rz 79.41 deg; joints [26.784, -65.118, 73.142, -8.884, 37.333, -89.386]
  MoveJ (Pt 7 (S135)) to (-479.15, -765.67, 391.59) mm, rotated rx 180 ry 0.34 rz 89.87 deg; joints [38.044, -66.874, 59.759, 6.703, 38.126, -89.694]
  MoveJ (Pt 8 (S168)) to (-520.28, -802.24, 391.81) mm, rotated rx 180 ry 0.34 rz 89.87 deg; joints [38.28, -60.592, 50.44, 9.726, 38.353, -89.675]
  MoveJ (Pt 9 (S109)) to (-370.5, -902.58, 392.41) mm, rotated rx 180 ry 0.34 rz 89.87 deg; joints [50.012, -60.823, 50.732, 9.743, 50.085, -89.789]
  MoveJ (Pt 10 (S147)) to (-379.6, -965.89, 392.79) mm, rotated rx 180 ry 0.34 rz 89.87 deg; joints [52.117, -52.777, 37.808, 14.617, 52.182, -89.782]
  MoveJ (Pt 11 (S204)) to (-424.15, -993, 386.99) mm, rotated rx -179.85 ry 0.6 rz 89.42 deg; joints [51.045, -45.985, 26.713, 18.574, 51.562, -89.705]
  MoveJ (Pt 12 (S233)) to (-323.88, -992.98, 486.72) mm, rotated rx -179.85 ry 0.6 rz 89.42 deg; joints [55.939, -45.623, 14.997, 29.967, 56.444, -89.768]
  MoveJ (Pt 13 (S232)) to (-432.46, -955.2, 486.62) mm, rotated rx -179.95 ry 0.62 rz 79.41 deg; joints [50.032, -46.238, 16.171, 29.419, 60.538, -89.707]

--- program bovenpickupToType13Instance17 (robot UR10e) ---
  MoveJ (Pt 1 (S537)) to (-569.02, 256.95, 231.44) mm, rotated rx 180 ry -0.01 rz 58.34 deg; joints [-50.868, -81.351, 94.607, -13.692, -19.23, -89.565]
  MoveJ (Pt 2 (S453)) to (-621.5, 171.83, 231.42) mm, rotated rx 180 ry -0.01 rz 58.34 deg; joints [-42.328, -81.409, 94.677, -14.057, -10.69, -89.211]
  MoveJ (Pt 3 (S393)) to (-700.22, 44.15, 231.39) mm, rotated rx 180 ry -0.01 rz 58.34 deg; joints [-29.369, -77.97, 90.586, -9.022, 2.264, -93.593]
  MoveJ (Pt 4 (S389)) to (-700.25, 44.11, 481.39) mm, rotated rx 180 ry -0.01 rz 58.34 deg; joints [-29.33, -78.074, 65.414, 15.651, 2.287, -92.99]
  MoveJ (Pt 5 (S369)) to (-619.87, -418.56, 481.52) mm, rotated rx -179.85 ry 0.6 rz 89.42 deg; joints [9.338, -76.474, 63.541, 10.042, 9.896, -87.311]
  MoveJ (Pt 6 (S464)) to (-570.29, -640.46, 483.71) mm, rotated rx -179.85 ry 0.6 rz 89.42 deg; joints [26.854, -67.916, 51.844, 14.953, 27.39, -89.171]
  MoveJ (Pt 7 (S675)) to (-370.28, -801.98, 491.81) mm, rotated rx 180 ry 0.34 rz 89.87 deg; joints [45.268, -68.448, 51.699, 16.383, 45.344, -89.76]
  MoveJ (Pt 8 (S801)) to (-279.38, -865.51, 492.19) mm, rotated rx 180 ry 0.34 rz 89.87 deg; joints [53.39, -66.86, 49.394, 17.137, 53.462, -89.821]
  MoveJ (Pt 9 (S881)) to (-170.5, -902.43, 492.41) mm, rotated rx 180 ry 0.34 rz 89.87 deg; joints [61.548, -67.173, 49.822, 17.048, 61.621, -89.875]
  MoveJ (Pt 10 (S919)) to (-124.99, -923.62, 485.44) mm, rotated rx -179.85 ry 0.6 rz 89.42 deg; joints [65.267, -66.64, 49.834, 16.228, 65.797, -89.935]

--- program bovenpickupToType13Instance18 (robot UR10e) ---
  MoveJ (Pt 1 (S552)) to (-569.02, 256.95, 231.44) mm, rotated rx 180 ry -0.01 rz 58.34 deg; joints [-50.868, -81.351, 94.607, -13.692, -19.23, -89.565]
  MoveJ (Pt 2 (S463)) to (-621.5, 171.83, 231.42) mm, rotated rx 180 ry -0.01 rz 58.34 deg; joints [-42.328, -81.409, 94.677, -14.057, -10.69, -89.211]
  MoveJ (Pt 3 (S385)) to (-700.22, 44.15, 231.39) mm, rotated rx 180 ry -0.01 rz 58.34 deg; joints [-29.369, -77.97, 90.586, -9.022, 2.264, -93.593]
  MoveJ (Pt 4 (S301)) to (-831.43, -168.65, 231.34) mm, rotated rx 180 ry -0.01 rz 58.34 deg; joints [-10.139, -68.333, 77.878, -9.215, 21.482, -90.324]
  MoveJ (Pt 5 (S475)) to (-570.99, -643.08, 233.72) mm, rotated rx -179.85 ry 0.6 rz 89.42 deg; joints [26.976, -69.099, 78.835, -10.802, 27.531, -89.229]
  MoveJ (Pt 6 (S530)) to (-378.82, -615.9, 390.7) mm, rotated rx 180 ry 0.34 rz 89.87 deg; joints [32.917, -85.112, 82.825, 1.871, 33.024, -89.684]
  MoveJ (Pt 7 (S681)) to (-270.06, -702.8, 391.22) mm, rotated rx 180 ry 0.34 rz 89.87 deg; joints [45.361, -84.322, 81.904, 2.087, 45.466, -89.81]
  MoveJ (Pt 8 (S992)) to (-20.28, -803.36, 391.82) mm, rotated rx 180 ry 0.34 rz 89.87 deg; joints [69.118, -82.29, 79.557, 2.458, 69.22, -89.954]
  MoveJ (Pt 9 (S1008)) to (-38.22, -879.93, 384.74) mm, rotated rx -179.85 ry 0.6 rz 89.42 deg; joints [70.042, -74.799, 71.224, 3.022, 70.59, -90.011]
  MoveJ (Pt 10 (S1088)) to (61.78, -880.95, 384.48) mm, rotated rx -179.85 ry 0.6 rz 89.42 deg; joints [77.61, -75.19, 71.751, 2.901, 78.159, -90.086]
  MoveJ (Pt 11 (S1090)) to (62.05, -879.9, 484.47) mm, rotated rx -179.85 ry 0.6 rz 89.42 deg; joints [77.626, -73.739, 59.711, 13.488, 78.165, -90.075]

--- program bovenpickupToType13Instance19 (robot UR10e) ---
  MoveJ (Pt 1 (S549)) to (-569.02, 256.95, 231.44) mm, rotated rx 180 ry -0.01 rz 58.34 deg; joints [-50.868, -81.351, 94.607, -13.692, -19.23, -89.565]
  MoveJ (Pt 2 (S464)) to (-621.5, 171.83, 231.42) mm, rotated rx 180 ry -0.01 rz 58.34 deg; joints [-42.328, -81.409, 94.677, -14.057, -10.69, -89.211]
  MoveJ (Pt 3 (S397)) to (-700.22, 44.15, 231.39) mm, rotated rx 180 ry -0.01 rz 58.34 deg; joints [-29.369, -77.97, 90.586, -9.022, 2.264, -93.593]
  MoveJ (Pt 4 (S392)) to (-700.25, 44.11, 481.39) mm, rotated rx 180 ry -0.01 rz 58.34 deg; joints [-29.33, -78.074, 65.414, 15.651, 2.287, -92.99]
  MoveJ (Pt 5 (S371)) to (-619.87, -418.56, 481.52) mm, rotated rx -179.85 ry 0.6 rz 89.42 deg; joints [9.338, -76.474, 63.541, 10.042, 9.896, -87.311]
  MoveJ (Pt 6 (S475)) to (-570.29, -640.46, 483.71) mm, rotated rx -179.85 ry 0.6 rz 89.42 deg; joints [26.854, -67.916, 51.844, 14.953, 27.39, -89.171]
  MoveJ (Pt 7 (S684)) to (-370.28, -801.98, 491.81) mm, rotated rx 180 ry 0.34 rz 89.87 deg; joints [45.268, -68.448, 51.699, 16.383, 45.344, -89.76]
  MoveJ (Pt 8 (S805)) to (-279.38, -865.51, 492.19) mm, rotated rx 180 ry 0.34 rz 89.87 deg; joints [53.39, -66.86, 49.394, 17.137, 53.462, -89.821]
  MoveJ (Pt 9 (S896)) to (-170.5, -902.43, 492.41) mm, rotated rx 180 ry 0.34 rz 89.87 deg; joints [61.548, -67.173, 49.822, 17.048, 61.621, -89.875]
  MoveJ (Pt 10 (S943)) to (-124.99, -923.62, 485.44) mm, rotated rx -179.85 ry 0.6 rz 89.42 deg; joints [65.267, -66.64, 49.834, 16.228, 65.797, -89.935]
  MoveJ (Pt 11 (S999)) to (-36.76, -953.12, 485.51) mm, rotated rx -179.85 ry 0.6 rz 89.42 deg; joints [71.94, -64.785, 47.115, 17.114, 72.467, -90.001]

--- program Type13Instance2Tobovenpickup (robot UR10e) ---
  MoveJ (Pt 1 (S1189)) to (-289.72, -617.57, 107.58) mm, rotated rx -88.79 ry -60.15 rz 178.37 deg; joints [27.28, -59.114, 114.207, 61.653, 76.16, 24.363]
  MoveJ (Pt 2 (S1201)) to (-339.48, -616.15, 194.31) mm, rotated rx -88.79 ry -60.15 rz 178.37 deg; joints [24.893, -63.386, 108.48, 72.156, 77.236, 22.181]
  MoveJ (Pt 3 (S1194)) to (-338.46, -516.17, 193.26) mm, rotated rx -88.79 ry -60.15 rz 178.37 deg; joints [14.894, -67.739, 116.253, 70.372, 81.948, 13.221]
  MoveJ (Pt 4 (S1230)) to (-326.21, -526.44, 274.18) mm, rotated rx -88.79 ry -60.15 rz 178.37 deg; joints [16.405, -73.929, 114.079, 78.537, 81.219, 14.568]
  MoveJ (Pt 5 (S1325)) to (-323.66, -276.47, 271.56) mm, rotated rx -88.79 ry -60.15 rz 178.37 deg; joints [-15.974, -82.156, 125.219, 76.084, 97.176, -13.671]
  MoveJ (Pt 6 (S1213)) to (-427.3, -109.3, 308.25) mm, rotated rx 88.03 ry -79.99 rz 1.82 deg; joints [-40.872, -92.425, 119.324, 55.78, 83.328, -40.3]
  MoveJ (Pt 7 (S1130)) to (-609.73, -107.84, 484.59) mm, rotated rx 89.55 ry -40 rz 0.16 deg; joints [-35.971, -95.179, 103.829, 37.546, 63.204, -24.789]
  MoveJ (Pt 8 (S396)) to (-575.98, -133.64, 570.37) mm, rotated rx 180 ry -0.01 rz 58.34 deg; joints [-28.022, -101.389, 88.85, 14.844, 3.631, -92.304]
  MoveJ (Pt 9 (S200)) to (-788.75, -2.39, 320.37) mm, rotated rx 180 ry -0.01 rz 58.34 deg; joints [-29.369, -77.97, 90.586, -9.022, 2.264, -93.593]
  MoveJ (Pt 10 (S218)) to (-710.03, 125.29, 320.4) mm, rotated rx 180 ry -0.01 rz 58.34 deg; joints [-42.328, -81.409, 94.677, -14.057, -10.69, -89.211]
  MoveJ (Pt 11 (S217)) to (-657.55, 210.41, 320.42) mm, rotated rx 180 ry -0.01 rz 58.34 deg; joints [-50.868, -81.351, 94.607, -13.692, -19.23, -89.565]

--- program Type13Instance3Tobovenpickup (robot UR10e) ---
  MoveJ (Pt 1 (S1294)) to (-267.62, -616.65, 217.16) mm, rotated rx 86.59 ry -79.83 rz 2.77 deg; joints [38.095, -81.767, 118.657, 44.846, 95.948, 38.281]
  MoveJ (Pt 2 (S1236)) to (-366.05, -615.46, 234.78) mm, rotated rx 86.59 ry -79.83 rz 2.77 deg; joints [30.962, -77.951, 111.623, 47.407, 94.864, 31.193]
  MoveJ (Pt 3 (S1190)) to (-428.42, -609.29, 311.25) mm, rotated rx 88.03 ry -79.99 rz 1.82 deg; joints [26.887, -78.117, 102.884, 56.217, 94.291, 26.679]
  MoveJ (Pt 4 (S1144)) to (-723.9, -523.05, 210.67) mm, rotated rx 86.59 ry -79.83 rz 2.77 deg; joints [10.723, -56.863, 83.085, 53.769, 91.432, 11.188]
  MoveJ (Pt 5 (S1130)) to (-718.8, -23.1, 205.42) mm, rotated rx 86.59 ry -79.83 rz 2.77 deg; joints [-30.172, -60.169, 89.434, 52.244, 84.533, -29.177]
  MoveJ (Pt 6 (S1084)) to (-609.73, -107.84, 484.59) mm, rotated rx 89.55 ry -40 rz 0.16 deg; joints [-35.971, -95.179, 103.829, 37.546, 63.204, -24.789]
  MoveJ (Pt 7 (S305)) to (-575.98, -133.64, 570.37) mm, rotated rx 180 ry -0.01 rz 58.34 deg; joints [-28.022, -101.389, 88.85, 14.844, 3.631, -92.304]
  MoveJ (Pt 8 (S158)) to (-788.75, -2.39, 320.37) mm, rotated rx 180 ry -0.01 rz 58.34 deg; joints [-29.369, -77.97, 90.586, -9.022, 2.264, -93.593]
  MoveJ (Pt 9 (S164)) to (-710.03, 125.29, 320.4) mm, rotated rx 180 ry -0.01 rz 58.34 deg; joints [-42.328, -81.409, 94.677, -14.057, -10.69, -89.211]
  MoveJ (Pt 10 (S161)) to (-657.55, 210.41, 320.42) mm, rotated rx 180 ry -0.01 rz 58.34 deg; joints [-50.868, -81.351, 94.607, -13.692, -19.23, -89.565]

--- program Type13Instance5Tobovenpickup (robot UR10e) ---
  MoveJ (Pt 1 (S133)) to (-131.68, -618.97, 128.27) mm, rotated rx -86.49 ry -80.13 rz 175.95 deg; joints [43.816, -74.655, 126.219, 45.161, 82.8, 43.896]
  MoveJ (Pt 2 (S93)) to (-230.2, -618.14, 111.17) mm, rotated rx -86.49 ry -80.13 rz 175.95 deg; joints [35.235, -69.52, 121.457, 45.798, 83.865, 35.319]
  MoveJ (Pt 3 (S77)) to (-247.29, -616.93, 209.69) mm, rotated rx -86.49 ry -80.13 rz 175.95 deg; joints [33.896, -76.471, 117.266, 57.083, 84.043, 33.995]
  MoveJ (Pt 4 (S75)) to (-348.42, -614.6, 333.21) mm, rotated rx 86.59 ry -79.83 rz 2.77 deg; joints [31.991, -83.698, 107.246, 57.617, 95.021, 32.221]
  MoveJ (Pt 5 (S49)) to (-428.42, -609.29, 311.25) mm, rotated rx 88.03 ry -79.99 rz 1.82 deg; joints [26.887, -78.117, 102.884, 56.217, 94.291, 26.679]
  MoveJ (Pt 6 (S13)) to (-723.9, -523.05, 210.67) mm, rotated rx 86.59 ry -79.83 rz 2.77 deg; joints [10.723, -56.863, 83.085, 53.769, 91.432, 11.188]
  MoveJ (Pt 7 (S99)) to (-718.8, -23.1, 205.42) mm, rotated rx 86.59 ry -79.83 rz 2.77 deg; joints [-30.172, -60.169, 89.434, 52.244, 84.533, -29.177]
  MoveJ (Pt 8 (S327)) to (-609.73, -107.84, 484.59) mm, rotated rx 89.55 ry -40 rz 0.16 deg; joints [-35.971, -95.179, 103.829, 37.546, 63.204, -24.789]
  MoveJ (Pt 9 (S848)) to (-575.98, -133.64, 570.37) mm, rotated rx 180 ry -0.01 rz 58.34 deg; joints [-28.022, -101.389, 88.85, 14.844, 3.631, -92.304]
  MoveJ (Pt 10 (S877)) to (-788.75, -2.39, 320.37) mm, rotated rx 180 ry -0.01 rz 58.34 deg; joints [-29.369, -77.97, 90.586, -9.022, 2.264, -93.593]
  MoveJ (Pt 11 (S1076)) to (-710.03, 125.29, 320.4) mm, rotated rx 180 ry -0.01 rz 58.34 deg; joints [-42.328, -81.409, 94.677, -14.057, -10.69, -89.211]
  MoveJ (Pt 12 (S1159)) to (-657.55, 210.41, 320.42) mm, rotated rx 180 ry -0.01 rz 58.34 deg; joints [-50.868, -81.351, 94.607, -13.692, -19.23, -89.565]

--- program Type13Instance6Tobovenpickup (robot UR10e) ---
  MoveJ (Pt 1 (S1552)) to (64.03, -619.93, 226.49) mm, rotated rx 86.59 ry -79.83 rz 2.77 deg; joints [79.719, -85.604, 123.467, 49.881, 100.002, 80.15]
  MoveJ (Pt 2 (S1551)) to (63.98, -610.91, 224.43) mm, rotated rx 88.03 ry -79.99 rz 1.82 deg; joints [79.127, -86.375, 124.464, 49.756, 99.857, 79.091]
  MoveJ (Pt 3 (S1550)) to (-67.18, -610.75, 202.29) mm, rotated rx 89.47 ry -50 rz 0.28 deg; joints [74.524, -83.635, 127.662, 33.189, 128.314, 70.315]
  MoveJ (Pt 4 (S1528)) to (-143.56, -510.2, 265.96) mm, rotated rx 89.47 ry -50 rz 0.28 deg; joints [52.736, -103.918, 134.566, 32.325, 120.747, 45.438]
  MoveJ (Pt 5 (S1495)) to (-322.41, -359.68, 284.88) mm, rotated rx 89.47 ry -50 rz 0.28 deg; joints [-10.312, -118.158, 138.236, 30.476, 83.322, -7.663]
  MoveJ (Pt 6 (S1259)) to (-609.73, -107.84, 484.59) mm, rotated rx 89.55 ry -40 rz 0.16 deg; joints [-35.971, -95.179, 103.829, 37.546, 63.204, -24.789]
  MoveJ (Pt 7 (S659)) to (-575.98, -133.64, 570.37) mm, rotated rx 180 ry -0.01 rz 58.34 deg; joints [-28.022, -101.389, 88.85, 14.844, 3.631, -92.304]
  MoveJ (Pt 8 (S426)) to (-788.75, -2.39, 320.37) mm, rotated rx 180 ry -0.01 rz 58.34 deg; joints [-29.369, -77.97, 90.586, -9.022, 2.264, -93.593]
  MoveJ (Pt 9 (S464)) to (-710.03, 125.29, 320.4) mm, rotated rx 180 ry -0.01 rz 58.34 deg; joints [-42.328, -81.409, 94.677, -14.057, -10.69, -89.211]
  MoveJ (Pt 10 (S461)) to (-657.55, 210.41, 320.42) mm, rotated rx 180 ry -0.01 rz 58.34 deg; joints [-50.868, -81.351, 94.607, -13.692, -19.23, -89.565]

--- program Type13Instance7Tobovenpickup (robot UR10e) ---
  MoveJ (Pt 1 (S149)) to (88.68, -622.23, 31.67) mm, rotated rx -89.21 ry -40.15 rz 178.91 deg; joints [54.508, -52.127, 132.503, 43.528, 51.005, 42.429]
  MoveJ (Pt 2 (S80)) to (-52.22, -620.92, 19.72) mm, rotated rx -89.21 ry -40.15 rz 178.91 deg; joints [39.475, -48.224, 127.844, 52.459, 60.292, 28.076]
  MoveJ (Pt 3 (S40)) to (-239.96, -618.99, 20.85) mm, rotated rx -88.79 ry -60.15 rz 178.37 deg; joints [30.052, -53.136, 118.304, 50.936, 74.933, 26.918]
  MoveJ (Pt 4 (S14)) to (-376.45, -617.21, 57.82) mm, rotated rx -88.79 ry -60.15 rz 178.37 deg; joints [23.502, -51.15, 106.698, 61.979, 77.87, 20.902]
  MoveJ (Pt 5 (S60)) to (-624.3, -614.84, 42.76) mm, rotated rx -86.49 ry -80.13 rz 175.95 deg; joints [18.033, -44.355, 85.466, 58.113, 86.348, 18.222]
  MoveJ (Pt 6 (S76)) to (-723.9, -523.05, 210.67) mm, rotated rx 86.59 ry -79.83 rz 2.77 deg; joints [10.723, -56.863, 83.085, 53.769, 91.432, 11.188]
  MoveJ (Pt 7 (S173)) to (-718.8, -23.1, 205.42) mm, rotated rx 86.59 ry -79.83 rz 2.77 deg; joints [-30.172, -60.169, 89.434, 52.244, 84.533, -29.177]
  MoveJ (Pt 8 (S190)) to (-609.73, -107.84, 484.59) mm, rotated rx 89.55 ry -40 rz 0.16 deg; joints [-35.971, -95.179, 103.829, 37.546, 63.204, -24.789]
  MoveJ (Pt 9 (S938)) to (-575.98, -133.64, 570.37) mm, rotated rx 180 ry -0.01 rz 58.34 deg; joints [-28.022, -101.389, 88.85, 14.844, 3.631, -92.304]
  MoveJ (Pt 10 (S960)) to (-788.75, -2.39, 320.37) mm, rotated rx 180 ry -0.01 rz 58.34 deg; joints [-29.369, -77.97, 90.586, -9.022, 2.264, -93.593]
  MoveJ (Pt 11 (S1072)) to (-710.03, 125.29, 320.4) mm, rotated rx 180 ry -0.01 rz 58.34 deg; joints [-42.328, -81.409, 94.677, -14.057, -10.69, -89.211]
  MoveJ (Pt 12 (S1133)) to (-657.55, 210.41, 320.42) mm, rotated rx 180 ry -0.01 rz 58.34 deg; joints [-50.868, -81.351, 94.607, -13.692, -19.23, -89.565]

--- program Type13Instance8Tobovenpickup (robot UR10e) ---
  MoveJ (Pt 1 (S133)) to (-385.19, -699.16, 372.43) mm, rotated rx -179.78 ry 45.6 rz 89.57 deg; joints [27.437, -91.84, 132.735, -106.178, 51.694, -36.835]
  MoveJ (Pt 2 (S138)) to (-438.23, -721.07, 395.91) mm, rotated rx 180 ry 45.34 rz 89.87 deg; joints [26.844, -88.33, 126.117, -103.53, 51.12, -35.687]
  MoveJ (Pt 3 (S174)) to (-425.45, -756.99, 432.24) mm, rotated rx 180 ry 45.34 rz 89.87 deg; joints [30.527, -89.213, 121.956, -95.887, 52.71, -39.909]
  MoveJ (Pt 4 (S192)) to (-385.14, -764.67, 439.92) mm, rotated rx 180 ry 45.34 rz 89.87 deg; joints [33.25, -91.757, 123.172, -92.767, 53.974, -42.917]
  MoveJ (Pt 5 (S285)) to (-385.37, -870.1, 546.62) mm, rotated rx 180 ry 45.34 rz 89.87 deg; joints [41.069, -88.108, 106.775, -75.506, 58, -50.992]
  MoveJ (Pt 6 (S626)) to (-385.77, -1045.81, 724.45) mm, rotated rx 180 ry 45.34 rz 89.87 deg; joints [50.594, -75.677, 73.548, -50.385, 63.524, -59.847]
  MoveJ (Pt 7 (S967)) to (-321.4, -888.21, 481.33) mm, rotated rx 180 ry 0.34 rz 89.87 deg; joints [50.999, -75.487, 71.344, 3.823, 51.092, -89.834]
  MoveJ (Pt 8 (S943)) to (-421.18, -787.99, 480.73) mm, rotated rx 180 ry 0.34 rz 89.87 deg; joints [39.494, -78.996, 75.747, 2.876, 39.592, -89.745]
  MoveJ (Pt 9 (S939)) to (-570.84, -637.66, 479.83) mm, rotated rx 180 ry 0.34 rz 89.87 deg; joints [22.274, -79.112, 75.978, 2.531, 22.373, -89.461]
  MoveJ (Pt 10 (S920)) to (-622.54, -727.68, 323.76) mm, rotated rx -179.85 ry 0.6 rz 89.42 deg; joints [26.976, -69.099, 78.835, -10.802, 27.531, -89.229]
  MoveJ (Pt 11 (S842)) to (-919.96, -215.19, 320.32) mm, rotated rx 180 ry -0.01 rz 58.34 deg; joints [-10.139, -68.333, 77.878, -9.215, 21.482, -90.324]
  MoveJ (Pt 12 (S781)) to (-788.75, -2.39, 320.37) mm, rotated rx 180 ry -0.01 rz 58.34 deg; joints [-29.369, -77.97, 90.586, -9.022, 2.264, -93.593]
  MoveJ (Pt 13 (S715)) to (-710.03, 125.29, 320.4) mm, rotated rx 180 ry -0.01 rz 58.34 deg; joints [-42.328, -81.409, 94.677, -14.057, -10.69, -89.211]
  MoveJ (Pt 14 (S719)) to (-657.55, 210.41, 320.42) mm, rotated rx 180 ry -0.01 rz 58.34 deg; joints [-50.868, -81.351, 94.607, -13.692, -19.23, -89.565]

--- program Type13Instance10Tobovenpickup (robot UR10e) ---
  MoveJ (Pt 1 (S289)) to (-188.6, -727.86, 399.15) mm, rotated rx -179.78 ry 45.6 rz 89.57 deg; joints [44.179, -104.134, 137.124, -88.349, 60.047, -54.438]
  MoveJ (Pt 2 (S334)) to (-134.98, -694.94, 368.79) mm, rotated rx 180 ry 45.34 rz 89.87 deg; joints [46.017, -108.293, 143.092, -89.199, 60.781, -55.795]
  MoveJ (Pt 3 (S487)) to (-88.08, -650.72, 466.2) mm, rotated rx 180 ry 45.34 rz 89.87 deg; joints [46.59, -123.031, 139.305, -70.413, 61.141, -56.34]
  MoveJ (Pt 4 (S556)) to (-62.19, -645.32, 440.42) mm, rotated rx -179.78 ry 45.6 rz 89.57 deg; joints [49.872, -123.512, 142.123, -71.486, 63.406, -59.701]
  MoveJ (Pt 5 (S900)) to (14.21, -469.79, 69.28) mm, rotated rx -179.85 ry 0.6 rz 89.42 deg; joints [50.086, -118.746, 152.354, -34.198, 50.72, -89.874]
  MoveJ (Pt 6 (S751)) to (-172.83, -513.5, 70.26) mm, rotated rx -179.85 ry 0.6 rz 89.42 deg; joints [29.31, -103.236, 144.185, -41.809, 29.916, -89.469]
  MoveJ (Pt 7 (S617)) to (-370.7, -482.88, 70.48) mm, rotated rx -179.85 ry 0.6 rz 89.42 deg; joints [13.149, -90.207, 133.323, -44.907, 13.74, -88.44]
  MoveJ (Pt 8 (S631)) to (-575.95, -133.6, 320.37) mm, rotated rx 180 ry -0.01 rz 58.34 deg; joints [-28.099, -101.276, 114.057, -10.072, 3.57, -92.709]
  MoveJ (Pt 9 (S658)) to (-624.91, 72.81, 320.4) mm, rotated rx 180 ry -0.01 rz 58.34 deg; joints [-44.286, -90.997, 104.968, -14.694, -12.634, -89.275]
  MoveJ (Pt 10 (S644)) to (-710.03, 125.29, 320.4) mm, rotated rx 180 ry -0.01 rz 58.34 deg; joints [-42.328, -81.409, 94.677, -14.057, -10.69, -89.211]
  MoveJ (Pt 11 (S728)) to (-657.55, 210.41, 320.42) mm, rotated rx 180 ry -0.01 rz 58.34 deg; joints [-50.868, -81.351, 94.607, -13.692, -19.23, -89.565]

--- program Type13Instance12Tobovenpickup (robot UR10e) ---
  MoveJ (Pt 1 (S513)) to (-12.15, -719.18, 387.98) mm, rotated rx -179.78 ry 45.6 rz 89.57 deg; joints [63.878, -109.293, 140.39, -79.57, 72.279, -71.376]
  MoveJ (Pt 2 (S634)) to (61.77, -722.18, 395.92) mm, rotated rx 180 ry 45.34 rz 89.87 deg; joints [74.106, -108.805, 138.636, -76.185, 78.931, -78.761]
  MoveJ (Pt 3 (S633)) to (61.39, -730.41, 398.49) mm, rotated rx -179.78 ry 45.6 rz 89.57 deg; joints [74.725, -107.766, 137.885, -76.607, 79.613, -79.609]
  MoveJ (Pt 4 (S805)) to (105.76, -665.07, 458.39) mm, rotated rx -179.78 ry 45.6 rz 89.57 deg; joints [79.214, -118.718, 137.07, -64.344, 82.733, -82.897]
  MoveJ (Pt 5 (S925)) to (129.27, -487.99, 69.16) mm, rotated rx -179.85 ry 0.6 rz 89.42 deg; joints [80.537, -109.201, 147.969, -39.291, 81.151, -90.195]
  MoveJ (Pt 6 (S723)) to (-84.6, -543.01, 70.32) mm, rotated rx -179.85 ry 0.6 rz 89.42 deg; joints [44.503, -103.995, 144.682, -41.32, 45.11, -89.793]
  MoveJ (Pt 7 (S709)) to (-172.83, -513.5, 70.26) mm, rotated rx -179.85 ry 0.6 rz 89.42 deg; joints [29.31, -103.236, 144.185, -41.809, 29.916, -89.469]
  MoveJ (Pt 8 (S570)) to (-370.7, -482.88, 70.48) mm, rotated rx -179.85 ry 0.6 rz 89.42 deg; joints [13.149, -90.207, 133.323, -44.907, 13.74, -88.44]
  MoveJ (Pt 9 (S757)) to (-575.95, -133.6, 320.37) mm, rotated rx 180 ry -0.01 rz 58.34 deg; joints [-28.099, -101.276, 114.057, -10.072, 3.57, -92.709]
  MoveJ (Pt 10 (S706)) to (-624.91, 72.81, 320.4) mm, rotated rx 180 ry -0.01 rz 58.34 deg; joints [-44.286, -90.997, 104.968, -14.694, -12.634, -89.275]
  MoveJ (Pt 11 (S716)) to (-710.03, 125.29, 320.4) mm, rotated rx 180 ry -0.01 rz 58.34 deg; joints [-42.328, -81.409, 94.677, -14.057, -10.69, -89.211]
  MoveJ (Pt 12 (S755)) to (-657.55, 210.41, 320.42) mm, rotated rx 180 ry -0.01 rz 58.34 deg; joints [-50.868, -81.351, 94.607, -13.692, -19.23, -89.565]

--- program Type13Instance13Tobovenpickup (robot UR10e) ---
  MoveJ (Pt 1 (S612)) to (56.33, -667.94, 334.76) mm, rotated rx -179.78 ry 45.6 rz 89.57 deg; joints [70.982, -111.414, 147.715, -83.342, 77.05, -76.836]
  MoveJ (Pt 2 (S623)) to (61.39, -730.41, 398.49) mm, rotated rx -179.78 ry 45.6 rz 89.57 deg; joints [74.725, -107.766, 137.885, -76.607, 79.613, -79.609]
  MoveJ (Pt 3 (S799)) to (105.76, -665.07, 458.39) mm, rotated rx -179.78 ry 45.6 rz 89.57 deg; joints [79.214, -118.718, 137.07, -64.344, 82.733, -82.897]
  MoveJ (Pt 4 (S942)) to (129.27, -487.99, 69.16) mm, rotated rx -179.85 ry 0.6 rz 89.42 deg; joints [80.537, -109.201, 147.969, -39.291, 81.151, -90.195]
  MoveJ (Pt 5 (S777)) to (-84.6, -543.01, 70.32) mm, rotated rx -179.85 ry 0.6 rz 89.42 deg; joints [44.503, -103.995, 144.682, -41.32, 45.11, -89.793]
  MoveJ (Pt 6 (S768)) to (-172.83, -513.5, 70.26) mm, rotated rx -179.85 ry 0.6 rz 89.42 deg; joints [29.31, -103.236, 144.185, -41.809, 29.916, -89.469]
  MoveJ (Pt 7 (S651)) to (-370.7, -482.88, 70.48) mm, rotated rx -179.85 ry 0.6 rz 89.42 deg; joints [13.149, -90.207, 133.323, -44.907, 13.74, -88.44]
  MoveJ (Pt 8 (S852)) to (-575.95, -133.6, 320.37) mm, rotated rx 180 ry -0.01 rz 58.34 deg; joints [-28.099, -101.276, 114.057, -10.072, 3.57, -92.709]
  MoveJ (Pt 9 (S802)) to (-624.91, 72.81, 320.4) mm, rotated rx 180 ry -0.01 rz 58.34 deg; joints [-44.286, -90.997, 104.968, -14.694, -12.634, -89.275]
  MoveJ (Pt 10 (S807)) to (-710.03, 125.29, 320.4) mm, rotated rx 180 ry -0.01 rz 58.34 deg; joints [-42.328, -81.409, 94.677, -14.057, -10.69, -89.211]
  MoveJ (Pt 11 (S809)) to (-657.55, 210.41, 320.42) mm, rotated rx 180 ry -0.01 rz 58.34 deg; joints [-50.868, -81.351, 94.607, -13.692, -19.23, -89.565]

--- program Type13Instance14Tobovenpickup (robot UR10e) ---
  MoveJ (Pt 1 (S656)) to (73.98, -766.28, 434.94) mm, rotated rx -179.78 ry 45.6 rz 89.57 deg; joints [77.62, -105.311, 132.061, -72.899, 81.611, -81.723]
  MoveJ (Pt 2 (S570)) to (61.39, -730.41, 398.49) mm, rotated rx -179.78 ry 45.6 rz 89.57 deg; joints [74.725, -107.766, 137.885, -76.607, 79.613, -79.609]
  MoveJ (Pt 3 (S750)) to (105.76, -665.07, 458.39) mm, rotated rx -179.78 ry 45.6 rz 89.57 deg; joints [79.214, -118.718, 137.07, -64.344, 82.733, -82.897]
  MoveJ (Pt 4 (S864)) to (129.27, -487.99, 69.16) mm, rotated rx -179.85 ry 0.6 rz 89.42 deg; joints [80.537, -109.201, 147.969, -39.291, 81.151, -90.195]
  MoveJ (Pt 5 (S664)) to (-84.6, -543.01, 70.32) mm, rotated rx -179.85 ry 0.6 rz 89.42 deg; joints [44.503, -103.995, 144.682, -41.32, 45.11, -89.793]
  MoveJ (Pt 6 (S644)) to (-172.83, -513.5, 70.26) mm, rotated rx -179.85 ry 0.6 rz 89.42 deg; joints [29.31, -103.236, 144.185, -41.809, 29.916, -89.469]
  MoveJ (Pt 7 (S579)) to (-370.7, -482.88, 70.48) mm, rotated rx -179.85 ry 0.6 rz 89.42 deg; joints [13.149, -90.207, 133.323, -44.907, 13.74, -88.44]
  MoveJ (Pt 8 (S770)) to (-575.95, -133.6, 320.37) mm, rotated rx 180 ry -0.01 rz 58.34 deg; joints [-28.099, -101.276, 114.057, -10.072, 3.57, -92.709]
  MoveJ (Pt 9 (S728)) to (-624.91, 72.81, 320.4) mm, rotated rx 180 ry -0.01 rz 58.34 deg; joints [-44.286, -90.997, 104.968, -14.694, -12.634, -89.275]
  MoveJ (Pt 10 (S814)) to (-710.03, 125.29, 320.4) mm, rotated rx 180 ry -0.01 rz 58.34 deg; joints [-42.328, -81.409, 94.677, -14.057, -10.69, -89.211]
  MoveJ (Pt 11 (S817)) to (-657.55, 210.41, 320.42) mm, rotated rx 180 ry -0.01 rz 58.34 deg; joints [-50.868, -81.351, 94.607, -13.692, -19.23, -89.565]

--- program Type13Instance15Tobovenpickup (robot UR10e) ---
  MoveJ (Pt 1 (S339)) to (-322.86, -892.99, 485.67) mm, rotated rx -179.85 ry 0.6 rz 89.42 deg; joints [51.242, -75.215, 70.66, 3.908, 51.792, -89.787]
  MoveJ (Pt 2 (S307)) to (-330.28, -851.53, 481.11) mm, rotated rx 180 ry 0.34 rz 89.87 deg; joints [48.532, -78.392, 74.978, 3.089, 48.628, -89.822]
  MoveJ (Pt 3 (S206)) to (-421.18, -787.99, 480.73) mm, rotated rx 180 ry 0.34 rz 89.87 deg; joints [39.494, -78.996, 75.747, 2.876, 39.592, -89.745]
  MoveJ (Pt 4 (S80)) to (-570.29, -640.46, 483.71) mm, rotated rx -179.85 ry 0.6 rz 89.42 deg; joints [22.508, -79.344, 75.967, 2.131, 23.068, -89.026]
  MoveJ (Pt 5 (S110)) to (-622.54, -727.68, 323.76) mm, rotated rx -179.85 ry 0.6 rz 89.42 deg; joints [26.976, -69.099, 78.835, -10.802, 27.531, -89.229]
  MoveJ (Pt 6 (S55)) to (-919.96, -215.19, 320.32) mm, rotated rx 180 ry -0.01 rz 58.34 deg; joints [-10.139, -68.333, 77.878, -9.215, 21.482, -90.324]
  MoveJ (Pt 7 (S70)) to (-788.75, -2.39, 320.37) mm, rotated rx 180 ry -0.01 rz 58.34 deg; joints [-29.369, -77.97, 90.586, -9.022, 2.264, -93.593]
  MoveJ (Pt 8 (S104)) to (-710.03, 125.29, 320.4) mm, rotated rx 180 ry -0.01 rz 58.34 deg; joints [-42.328, -81.409, 94.677, -14.057, -10.69, -89.211]
  MoveJ (Pt 9 (S159)) to (-657.55, 210.41, 320.42) mm, rotated rx 180 ry -0.01 rz 58.34 deg; joints [-50.868, -81.351, 94.607, -13.692, -19.23, -89.565]

--- program Type13Instance16Tobovenpickup (robot UR10e) ---
  MoveJ (Pt 1 (S641)) to (-432.46, -955.2, 486.62) mm, rotated rx -179.95 ry 0.62 rz 79.41 deg; joints [50.203, -65.499, 57.33, 7.549, 60.74, -89.765]
  MoveJ (Pt 2 (S593)) to (-430.5, -951.3, 481.71) mm, rotated rx 180 ry 0.34 rz 89.87 deg; joints [47.928, -64.077, 55.644, 8.081, 48.005, -89.782]
  MoveJ (Pt 3 (S498)) to (-421.4, -887.99, 481.33) mm, rotated rx 180 ry 0.34 rz 89.87 deg; joints [45.289, -70.532, 64.83, 5.348, 45.375, -89.777]
  MoveJ (Pt 4 (S476)) to (-530.28, -851.08, 481.11) mm, rotated rx 180 ry 0.34 rz 89.87 deg; joints [38.044, -66.874, 59.759, 6.703, 38.126, -89.694]
  MoveJ (Pt 5 (S248)) to (-698.6, -740.46, 324.1) mm, rotated rx -179.95 ry 0.62 rz 79.41 deg; joints [26.784, -65.118, 73.142, -8.884, 37.333, -89.386]
  MoveJ (Pt 6 (S24)) to (-622.54, -727.68, 323.76) mm, rotated rx -179.85 ry 0.6 rz 89.42 deg; joints [26.976, -69.099, 78.835, -10.802, 27.531, -89.229]
  MoveJ (Pt 7 (S180)) to (-919.96, -215.19, 320.32) mm, rotated rx 180 ry -0.01 rz 58.34 deg; joints [-10.139, -68.333, 77.878, -9.215, 21.482, -90.324]
  MoveJ (Pt 8 (S363)) to (-788.75, -2.39, 320.37) mm, rotated rx 180 ry -0.01 rz 58.34 deg; joints [-29.369, -77.97, 90.586, -9.022, 2.264, -93.593]
  MoveJ (Pt 9 (S405)) to (-710.03, 125.29, 320.4) mm, rotated rx 180 ry -0.01 rz 58.34 deg; joints [-42.328, -81.409, 94.677, -14.057, -10.69, -89.211]
  MoveJ (Pt 10 (S481)) to (-657.55, 210.41, 320.42) mm, rotated rx 180 ry -0.01 rz 58.34 deg; joints [-50.868, -81.351, 94.607, -13.692, -19.23, -89.565]

--- program Type13Instance17Tobovenpickup (robot UR10e) ---
  MoveJ (Pt 1 (S654)) to (-124.99, -923.62, 485.44) mm, rotated rx -179.85 ry 0.6 rz 89.42 deg; joints [66.188, -78.303, 74.533, 3.209, 66.741, -89.976]
  MoveJ (Pt 2 (S587)) to (-315.79, -875.28, 485.47) mm, rotated rx -179.95 ry 0.62 rz 79.41 deg; joints [53.381, -78.315, 74.551, 3.172, 63.935, -89.83]
  MoveJ (Pt 3 (S501)) to (-330.28, -851.53, 481.11) mm, rotated rx 180 ry 0.34 rz 89.87 deg; joints [48.532, -78.392, 74.978, 3.089, 48.628, -89.822]
  MoveJ (Pt 4 (S442)) to (-421.18, -787.99, 480.73) mm, rotated rx 180 ry 0.34 rz 89.87 deg; joints [39.494, -78.996, 75.747, 2.876, 39.592, -89.745]
  MoveJ (Pt 5 (S269)) to (-570.29, -640.46, 483.71) mm, rotated rx -179.85 ry 0.6 rz 89.42 deg; joints [22.508, -79.344, 75.967, 2.131, 23.068, -89.026]
  MoveJ (Pt 6 (S286)) to (-622.54, -727.68, 323.76) mm, rotated rx -179.85 ry 0.6 rz 89.42 deg; joints [26.976, -69.099, 78.835, -10.802, 27.531, -89.229]
  MoveJ (Pt 7 (S341)) to (-919.96, -215.19, 320.32) mm, rotated rx 180 ry -0.01 rz 58.34 deg; joints [-10.139, -68.333, 77.878, -9.215, 21.482, -90.324]
  MoveJ (Pt 8 (S383)) to (-788.75, -2.39, 320.37) mm, rotated rx 180 ry -0.01 rz 58.34 deg; joints [-29.369, -77.97, 90.586, -9.022, 2.264, -93.593]
  MoveJ (Pt 9 (S422)) to (-710.03, 125.29, 320.4) mm, rotated rx 180 ry -0.01 rz 58.34 deg; joints [-42.328, -81.409, 94.677, -14.057, -10.69, -89.211]
  MoveJ (Pt 10 (S468)) to (-657.55, 210.41, 320.42) mm, rotated rx 180 ry -0.01 rz 58.34 deg; joints [-50.868, -81.351, 94.607, -13.692, -19.23, -89.565]

--- program Type13Instance18Tobovenpickup (robot UR10e) ---
  MoveJ (Pt 1 (S720)) to (62.05, -879.9, 484.47) mm, rotated rx -179.85 ry 0.6 rz 89.42 deg; joints [80.496, -83.347, 80.539, 2.274, 81.055, -90.126]
  MoveJ (Pt 2 (S584)) to (-37.94, -878.88, 484.74) mm, rotated rx -179.85 ry 0.6 rz 89.42 deg; joints [71.784, -83.671, 80.876, 2.251, 72.344, -90.042]
  MoveJ (Pt 3 (S506)) to (-71.4, -888.77, 481.33) mm, rotated rx 180 ry 0.34 rz 89.87 deg; joints [69.118, -82.29, 79.557, 2.458, 69.22, -89.954]
  MoveJ (Pt 4 (S121)) to (-321.18, -788.22, 480.73) mm, rotated rx 180 ry 0.34 rz 89.87 deg; joints [45.361, -84.322, 81.904, 2.087, 45.466, -89.81]
  MoveJ (Pt 5 (S91)) to (-429.94, -701.31, 480.21) mm, rotated rx 180 ry 0.34 rz 89.87 deg; joints [32.917, -85.112, 82.825, 1.871, 33.024, -89.684]
  MoveJ (Pt 6 (S68)) to (-622.54, -727.68, 323.76) mm, rotated rx -179.85 ry 0.6 rz 89.42 deg; joints [26.976, -69.099, 78.835, -10.802, 27.531, -89.229]
  MoveJ (Pt 7 (S39)) to (-919.96, -215.19, 320.32) mm, rotated rx 180 ry -0.01 rz 58.34 deg; joints [-10.139, -68.333, 77.878, -9.215, 21.482, -90.324]
  MoveJ (Pt 8 (S16)) to (-788.75, -2.39, 320.37) mm, rotated rx 180 ry -0.01 rz 58.34 deg; joints [-29.369, -77.97, 90.586, -9.022, 2.264, -93.593]
  MoveJ (Pt 9 (S32)) to (-710.03, 125.29, 320.4) mm, rotated rx 180 ry -0.01 rz 58.34 deg; joints [-42.328, -81.409, 94.677, -14.057, -10.69, -89.211]
  MoveJ (Pt 10 (S52)) to (-657.55, 210.41, 320.42) mm, rotated rx 180 ry -0.01 rz 58.34 deg; joints [-50.868, -81.351, 94.607, -13.692, -19.23, -89.565]

--- program Type13Instance19Tobovenpickup (robot UR10e) ---
  MoveJ (Pt 1 (S655)) to (-36.76, -953.12, 485.51) mm, rotated rx -179.85 ry 0.6 rz 89.42 deg; joints [73.751, -76.309, 72.059, 3.706, 74.301, -90.05]
  MoveJ (Pt 2 (S624)) to (-25, -924.64, 485.18) mm, rotated rx -179.85 ry 0.6 rz 89.42 deg; joints [74.025, -79.207, 75.653, 3.013, 74.578, -90.057]
  MoveJ (Pt 3 (S540)) to (-71.4, -888.77, 481.33) mm, rotated rx 180 ry 0.34 rz 89.87 deg; joints [69.118, -82.29, 79.557, 2.458, 69.22, -89.954]
  MoveJ (Pt 4 (S332)) to (-321.18, -788.22, 480.73) mm, rotated rx 180 ry 0.34 rz 89.87 deg; joints [45.361, -84.322, 81.904, 2.087, 45.466, -89.81]
  MoveJ (Pt 5 (S298)) to (-429.94, -701.31, 480.21) mm, rotated rx 180 ry 0.34 rz 89.87 deg; joints [32.917, -85.112, 82.825, 1.871, 33.024, -89.684]
  MoveJ (Pt 6 (S357)) to (-622.54, -727.68, 323.76) mm, rotated rx -179.85 ry 0.6 rz 89.42 deg; joints [26.976, -69.099, 78.835, -10.802, 27.531, -89.229]
  MoveJ (Pt 7 (S551)) to (-919.96, -215.19, 320.32) mm, rotated rx 180 ry -0.01 rz 58.34 deg; joints [-10.139, -68.333, 77.878, -9.215, 21.482, -90.324]
  MoveJ (Pt 8 (S647)) to (-788.75, -2.39, 320.37) mm, rotated rx 180 ry -0.01 rz 58.34 deg; joints [-29.369, -77.97, 90.586, -9.022, 2.264, -93.593]
  MoveJ (Pt 9 (S683)) to (-710.03, 125.29, 320.4) mm, rotated rx 180 ry -0.01 rz 58.34 deg; joints [-42.328, -81.409, 94.677, -14.057, -10.69, -89.211]
  MoveJ (Pt 10 (S760)) to (-657.55, 210.41, 320.42) mm, rotated rx 180 ry -0.01 rz 58.34 deg; joints [-50.868, -81.351, 94.607, -13.692, -19.23, -89.565]

--- program helicoil pickup (robot UR10e) ---
  Set Ref.: UR10e Base
  Set Tool: Screwdriver indraaitool
  MoveL (boven pick-up)
  Call retract shank
  MoveL (pick-up) [its target is no longer in the station]
  Call get_helicoil
  MoveL (unclamped)
  Call retract shank
  MoveL (boven pick-up)

--- Python program retract shank ---
from robodk import robolink, robomath
import time
import requests
RDK = robolink.Robolink()
robot = RDK.Item('UR10e')

# Screwdriver data
compute_box_ip = "192.168.12.15"
username = "admin"
password = "OnRobotPerron038"
tool_id = 0  # ID of the tool

#default parameters screwdriver
shaft_value = 0 #shaft position

# URL's for screwdriver commands
shank_url =  f"http://{compute_box_ip}/api/dc/sd/move_shank/{tool_id}/{shaft_value}"


#---Main Program---

#Retract shank
requests.get(shank_url, auth=(username, password))
time.sleep(1) # 1s delay
print('klaar')

--- Python program get_helicoil ---
from robodk import robolink, robomath
import time
import requests
RDK = robolink.Robolink()
robot = RDK.Item('UR10e')

DEBUG=True
if DEBUG:
    RDK.setRunMode(robolink.RUNMODE_RUN_ROBOT) #Programma wordt uitgevoerd op de robot wanneer afgespeeld vanuit de editor

#Screwdriver data
compute_box_ip = "192.168.12.15"
username = "admin"
password = "OnRobotPerron038"
tool_id = 0  # ID of the tool

#default parameters screwdriver
max_torque = .2 #max torque untill stopping screw motion via default premount behavior
screw_length = 20 #helicoil length
target_torque = 1 #target torque to stop the screw motion early via monitoring current torque and no shank motion
shank_force = 20 #shank force
shaft_value = 0

# URL's for screwdriver commands
tighten_url = f"http://{compute_box_ip}/api/dc/sd/tighten/{tool_id}/{shank_force}/{screw_length}/{max_torque}"
shank_url =  f"http://{compute_box_ip}/api/dc/sd/move_shank/{tool_id}/{shaft_value}"


#---Main Program---
print('main program')
helicoil_detect = robot.getDI(0) #output is een string: '0.000000' of '1.000000'

#get helicoil from stepfeeder
if helicoil_detect != '1.000000':
    #Move actuator
    robot.setDO(2, 1)
    robot.setDO(4, 0)
    time.sleep(4)
    #trigger feeder
    robot.setAO(0, 0.4)

#wait until helicoil is detected
helicoil_detect = robot.getDI(0)
while helicoil_detect != '1.000000':
    time.sleep(0.1)
    helicoil_detect = robot.getDI(0)

#stop feeder
robot.setAO(0, 0)

#move cylinder out
robot.setDO(2, 0)
robot.setDO(4, 1)
time.sleep(5)

#Screw on helicoil
requests.get(tighten_url, auth=(username, password))
time.sleep(3)
shaft_value=24
shank_url =  f"http://{compute_box_ip}/api/dc/sd/move_shank/{tool_id}/{shaft_value}"
requests.get(shank_url, auth=(username, password))
time.sleep(1)

#Unclamp helicoil
robot.setDO(4, 0)
robot.setDO(2, 1)
time.sleep(.1)
robot.setDO(2, 0)

--- Python program Insert helicoil ---
from robodk import robolink, robomath
import time
import requests
import tkinter as tk
from tkinter import messagebox

RDK = robolink.Robolink()
robot = RDK.Item('UR10e')

DEBUG=True
if DEBUG:
    RDK.setRunMode(robolink.RUNMODE_RUN_ROBOT) #Programma wordt uitgevoerd op de robot wanneer afgespeeld vanuit de editor

#Screwdriver data
compute_box_ip = "192.168.12.15"
username = "admin"
password = "OnRobotPerron038"
tool_id = 0  # ID of the tool

#default parameters screwdriver
shank_force = 20 #shank force
screw_length = 20 #helicoil length
max_torque = 1.5 #max torque untill stopping screw motion via default premount behavior
unscrewing_length_mm = 20
shaft_value = 0 #shank position

# URL's for screwdriver commands
tighten_url = f"http://{compute_box_ip}/api/dc/sd/tighten/{tool_id}/{shank_force}/{screw_length}/{max_torque}"
shank_url =  f"http://{compute_box_ip}/api/dc/sd/move_shank/{tool_id}/{shaft_value}"
unscrew_url = f"http://{compute_box_ip}/api/dc/sd/loosen/{tool_id}/{shank_force}/{unscrewing_length_mm}"

#---Main Program---
shaft_value = 10
shank_url =  f"http://{compute_box_ip}/api/dc/sd/move_shank/{tool_id}/{shaft_value}"
requests.get(shank_url, auth=(username, password))

root = tk.Tk()
root.withdraw()
messagebox.showinfo("Notification", "Is the tool well aligned with the hole?")
root.destroy()
time.sleep(5)


requests.get(tighten_url, auth=(username, password))
time.sleep(13)

requests.get(unscrew_url, auth=(username, password))
time.sleep(8)

shaft_value = 0
shank_url =  f"http://{compute_box_ip}/api/dc/sd/move_shank/{tool_id}/{shaft_value}"
requests.get(shank_url, auth=(username, password))
time.sleep(2)

--- Python program pickup helicoil ---
import tkinter as tk
from tkinter import messagebox

# Hide the main tkinter window
root = tk.Tk()
root.withdraw()

# Trigger the message box
messagebox.showinfo("Notification", "Is the helicoil screwed onto the tool?")

# Close the hidden window
root.destroy()

--- Python program Test get screwdriver data ---
from robodk import robolink, robomath
import time
import requests
RDK = robolink.Robolink()
robot = RDK.Item('UR10e')

DEBUG=True
if DEBUG:
    RDK.setRunMode(robolink.RUNMODE_RUN_ROBOT) #Programma wordt uitgevoerd op de robot wanneer afgespeeld vanuit de editor

#Screwdriver data
compute_box_ip = "192.168.12.15"
username = "admin"
password = "OnRobotPerron038"
tool_id = 0  # ID of the tool

#default parameters screwdriver
shank_force = 20 #shank force
screw_length = 18 #helicoil length
max_torque = 1.5 #max torque untill stopping screw motion via default premount behavior
unscrewing_length_mm = 20
shaft_value = 0 #shank position

# URL's for screwdriver commands
tighten_url = f"http://{compute_box_ip}/api/dc/sd/tighten/{tool_id}/{shank_force}/{screw_length}/{max_torque}"
shank_url =  f"http://{compute_box_ip}/api/dc/sd/move_shank/{tool_id}/{shaft_value}"
unscrew_url = f"http://{compute_box_ip}/api/dc/sd/loosen/{tool_id}/{shank_force}/{unscrewing_length_mm}"

# URL's to get screwdriver data
busy_url = f"http://{compute_box_ip}/api/dc/sd/status/{tool_id}"


#---Main Program---
response = requests.get(busy_url, auth=(username, password))
print(response)
